	fb103StartQuiescentMode.ipDALICommunication := ipDALICommunication;
	fb103StopQuiescentMode.ipDALICommunication := ipDALICommunication;
	fb208QueryGearType.ipDALICommunication := ipDALICommunication;
	fb208QueryFeatures.ipDALICommunication := ipDALICommunication;
	fb208QuerySwitchStatus.ipDALICommunication := ipDALICommunication;
	fb208QueryDownSwitchOffThreshold.ipDALICommunication := ipDALICommunication;
	fb208QueryDownSwitchOnThreshold.ipDALICommunication := ipDALICommunication;
	fb208QueryUpSwitchOffThreshold.ipDALICommunication := ipDALICommunication;
	fb208QueryUpSwitchOnThreshold.ipDALICommunication := ipDALICommunication;
	fb208SetDownSwitchOffThreshold.ipDALICommunication := ipDALICommunication;
	fb208SetDownSwitchOnThreshold.ipDALICommunication := ipDALICommunication;
	fb208SetUpSwitchOffThreshold.ipDALICommunication := ipDALICommunication;
	fb208SetUpSwitchOnThreshold.ipDALICommunication := ipDALICommunication;
{endregion}
{region "Read"}
5:
{region "Start Qiescent Mode"}
	fb103StartQuiescentMode(bStart := TRUE,
							eAddressType := Tc3_DALI.E_DALIAddressType.Broadcast,
							eCommandPriority := Tc3_DALI.E_DALICommandPriority.Middle);
	IF (NOT fb103StartQuiescentMode.bBusy) THEN
		fb103StartQuiescentMode(bStart := FALSE);
		nStep := 10;
	END_IF
{endregion}
10:
{region "Query Gear Type"}
	fb208QueryGearType(	bStart := TRUE,
						nAddress := nAddress,
						eAddressType := Tc3_DALI.E_DALIAddressType.Short,
						eCommandPriority := Tc3_DALI.E_DALICommandPriority.Middle,
						nGearType => nGearType);
	IF (NOT fb208QueryGearType.bBusy) THEN
		fb208QueryGearType(bStart := FALSE);
		sGearType := GearType(nGearType := nGearType);
		nStep := 20;
	END_IF
{endregion}
20:
{region "Query Features"}
	fb208QueryFeatures(	bStart := TRUE,
						nAddress := nAddress,
						eAddressType := Tc3_DALI.E_DALIAddressType.Short,
						eCommandPriority := Tc3_DALI.E_DALICommandPriority.Middle);
	IF (NOT fb208QueryFeatures.bBusy) THEN
		fb208QueryFeatures(bStart := FALSE);
		bThreshold := fb208QueryFeatures.nFeatures.3;
		bAddressingPhysical := fb208QueryFeatures.nFeatures.7;
		nStep := 30;
	END_IF
{endregion}
30:
{region "Query Down Switch Off Threshold"}
	fb208QueryDownSwitchOffThreshold(	bStart := TRUE,
										nAddress := nAddress,
										eAddressType := Tc3_DALI.E_DALIAddressType.Short,
										eCommandPriority := Tc3_DALI.E_DALICommandPriority.Middle);
	IF (NOT fb208QueryDownSwitchOffThreshold.bBusy) THEN
		fb208QueryDownSwitchOffThreshold(bStart := FALSE);
		nDownSwitchOffThreshold := fb208QueryDownSwitchOffThreshold.nDownSwitchOffThreshold;
		nStep := 40;
	END_IF
{endregion}
40:
{region "Query Down Switch On Threshold"}
	fb208QueryDownSwitchOnThreshold(bStart := TRUE,
									nAddress := nAddress,
									eAddressType := Tc3_DALI.E_DALIAddressType.Short,
									eCommandPriority := Tc3_DALI.E_DALICommandPriority.Middle);
	IF (NOT fb208QueryDownSwitchOnThreshold.bBusy) THEN
		fb208QueryDownSwitchOnThreshold(bStart := FALSE);
		nDownSwitchOnThreshold := fb208QueryDownSwitchOnThreshold.nDownSwitchOnThreshold;
		nStep := 50;
	END_IF
{endregion}
50:
{region "Query Up Switch Off Threshold"}
	fb208QueryUpSwitchOffThreshold(	bStart := TRUE,
									nAddress := nAddress,
									eAddressType := Tc3_DALI.E_DALIAddressType.Short,
									eCommandPriority := Tc3_DALI.E_DALICommandPriority.Middle);
	IF (NOT fb208QueryUpSwitchOffThreshold.bBusy) THEN
		fb208QueryUpSwitchOffThreshold(bStart := FALSE);
		nUpSwitchOffThreshold := fb208QueryUpSwitchOffThreshold.nUpSwitchOffThreshold;
		nStep := 60;
	END_IF
{endregion}
60:
{region "Query Up Switch On Threshold"}
	fb208QueryUpSwitchOnThreshold(	bStart := TRUE,
									nAddress := nAddress,
									eAddressType := Tc3_DALI.E_DALIAddressType.Short,
									eCommandPriority := Tc3_DALI.E_DALICommandPriority.Middle );
	IF (NOT fb208QueryUpSwitchOnThreshold.bBusy) THEN
		fb208QueryUpSwitchOnThreshold(bStart := FALSE);
		nUpSwitchOnThreshold := fb208QueryUpSwitchOnThreshold.nUpSwitchOnThreshold;
		nStep := 70;
	END_IF
{endregion}
70:
{region "Stop Qiescent Mode"}
	fb103StopQuiescentMode(	bStart := TRUE,
							eAddressType := Tc3_DALI.E_DALIAddressType.Broadcast,
							eCommandPriority := Tc3_DALI.E_DALICommandPriority.Middle);
	IF (NOT fb103StopQuiescentMode.bBusy) THEN
		fb103StopQuiescentMode(bStart:= FALSE);
		nStep := 0;
	END_IF
{endregion}
{region "Write"}
500:
{region "Set Down Switch Off Threshold"}
	fb208SetDownSwitchOffThreshold(	bStart := TRUE,
									nAddress := nAddress,
									eAddressType := Tc3_DALI.E_DALIAddressType.Short,
									eCommandPriority := Tc3_DALI.E_DALICommandPriority.Middle,
									nDownSwitchOffThreshold := nDownSwitchOffThreshold);
	IF (NOT fb208SetDownSwitchOffThreshold.bBusy) THEN
		fb208SetDownSwitchOffThreshold(bStart := FALSE);
		nStep := 510;
	END_IF
{endregion}
510:
{region "Set Down Switch On Threshold"}
	fb208SetDownSwitchOnThreshold(	bStart := TRUE,
									nAddress := nAddress,
									eAddressType := Tc3_DALI.E_DALIAddressType.Short,
									eCommandPriority := Tc3_DALI.E_DALICommandPriority.Middle,
									nDownSwitchOnThreshold := nDownSwitchOnThreshold);
	IF (NOT fb208SetDownSwitchOnThreshold.bBusy) THEN
		fb208SetDownSwitchOnThreshold(bStart := FALSE);
		nStep := 520;
	END_IF
{endregion}
520:
{region "Set Up Switch Off Threshold"}
	fb208SetUpSwitchOffThreshold(	bStart := TRUE,
									nAddress := nAddress,
									eAddressType := Tc3_DALI.E_DALIAddressType.Short,
									eCommandPriority := Tc3_DALI.E_DALICommandPriority.Middle,
									nUpSwitchOffThreshold := nUpSwitchOffThreshold);
	IF (NOT fb208SetUpSwitchOffThreshold.bBusy) THEN
		fb208SetUpSwitchOffThreshold(bStart := FALSE);
		nStep := 530;
	END_IF
{endregion}
530:
{region "Set Up Switch On Threshold"}
	fb208SetUpSwitchOnThreshold(bStart := TRUE,
								nAddress := nAddress,
								eAddressType := Tc3_DALI.E_DALIAddressType.Short,
								eCommandPriority := Tc3_DALI.E_DALICommandPriority.Middle,
								nUpSwitchOnThreshold := nUpSwitchOnThreshold);
	IF (NOT fb208SetUpSwitchOnThreshold.bBusy) THEN
		fb208SetUpSwitchOnThreshold(bStart := FALSE);
		nStep := 0;
	END_IF
{endregion}
{endregion}
END_CASE
{endregion}

END_FUNCTION_BLOCK

// ---- POUs/DALI/PRGs/EnergyData/P_DALI_Energy_Line.TcPOU
(*
EnergyReporting reads ActiveEnergy (part 252) for all present ballasts on all (configured) DALI-lines where GVL_DALI.g_arrEnergyData[*DALI-line*,*ballast*].bHasEnergyData is TRUE.
Results are stored in GVL_DALI.g_arrEnergyData[*DALI-line*,*ballast*].fActiveEnergy. Energy Data for individual ballasts is NOT persistent.
The engergy sum per DALI-Line (Wh) and Total Energy (kWh) are persistent.

If bCheckActiveEnergy is TRUE, all present ballasts are queried for ActiveEnergy and bHasEnergyData is updated accordingly.
This will result in errors for any ballast that does not comply with part 252.
Errors will not be triggered for activations where bCheckActiveEnergy is FALSE.

After shutdown or download to PLC EnergyReporting is activated automatically internally with bCheckActiveEnergy set to TRUE

EnergyReporting is activated automatically at TOD 0:00, 6:00, 12:00, 18:00 (configurable)

NB:	The priority of commands are set to "middle" internally. Updating all lines will take a couple of minutes to finish, so be patient.
	Other critical commands on the DALI-lines take priotity.
	Add appropriate communication immediately after configuration of a new KL6821 terminal.
	That is, arrfbDALI_EnergyReporting[*DALI-Line*].ipDALICommunication := P_DALI_Background.arrfbKL6821Communication[*DALI-Line*];
*)


PROGRAM P_DALI_Energy_Line
VAR
	arrfbDALI_EnergyReporting	: ARRAY[1..SH_Light.DALI_Param.MAX_DALIV2_LINES] OF FB_DALI_EnergyReporting;
	fbDALI_EnergyDataManagement	: SH_Light.FB_DALI_EnergyDataManagement;
	nNumOfEnergyLines			: BYTE;
	bReadEnergyDataAllLines		: BOOL;
	bReportingDone				: BOOL;
	fbRTrig_ReportingDone		: R_TRIG;
	bRTrigReportingDone			: BOOL;
	
	//Task scheduling
	stLocalSystemTime 		: TIMESTRUCT;
	fbLocalSystemTime 		: FB_LocalSystemTime;
	bGetTime 				: BOOL := TRUE;
	tTimeOut 				: TIME := DEFAULT_ADS_TIMEOUT;
	bLocalSystemTimeValid	: BOOL;
	tzID       				: E_TimeZoneID := eTimeZoneID_Invalid;
	
	tdSystemTime			: TOD;
	btestTodCompare			: BOOL;
	
	
END_VAR
VAR CONSTANT
	tdMidnight						: TOD := TOD#0:0:0;
	tdMorning						: TOD := TOD#6:0:0;
	tdMidDay						: TOD := TOD#12:0:0;
	tdEvening						: TOD := TOD#18:0:0;
	tCheckDuration					: TIME:= T#5S;
	tdTestsum						: TOD := (tdMidnight + tCheckDuration);
END_VAR

VAR PERSISTENT
	arrDaliLineEnergySumWh				: ARRAY[1..SH_Light.DALI_Param.MAX_DALIV2_LINES] OF LREAL;
	fTotalEnergyWh								: LREAL;
	nMaxControlGearOperatingHours		: UINT;
END_VAR


arrfbDALI_EnergyReporting[1].ipDALICommunication := P_DALI_Background.arrfbKL6821Communication[1];
arrfbDALI_EnergyReporting[2].ipDALICommunication := P_DALI_Background.arrfbKL6821Communication[2];
arrfbDALI_EnergyReporting[3].ipDALICommunication := P_DALI_Background.arrfbKL6821Communication[3];
//arrfbDALI_EnergyReporting[4].ipDALICommunication := P_DALI_Background.arrfbKL6821Communication[4];
//arrfbDALI_EnergyReporting[5].ipDALICommunication := P_DALI_Background.arrfbKL6821Communication[5];
//arrfbDALI_EnergyReporting[6].ipDALICommunication := P_DALI_Background.arrfbKL6821Communication[6]; // for more update SH_Light.DALI_Param.MAX_DALIV2_LINES

nNumOfEnergyLines := 3;

fbLocalSystemTime(
	sNetID:= '', 
	bEnable:= bGetTime, 
	dwCycle:= 2, // cycle time (in seconds) , Synchronization  every 2 seconds.
	dwOpt:= 1, //Bit 0: If this is set, the Windows system time is additionally synchronized cyclically with the hardware clock (RTC) (corresponds to the function NT_SetTimeToRTCTime).
	tTimeout:= tTimeOut, 
	bValid=> bLocalSystemTimeValid, 
	systemTime=> stLocalSystemTime, 
	tzID=> tzID);
	
tdSystemTime := SYSTEMTIME_TO_TOD(systemTime := stLocalSystemTime);
IF	((tdSystemTime > tdMidnight AND tdSystemTime < (tdMidnight + tCheckDuration)) OR (tdSystemTime > tdMorning AND tdSystemTime < (tdMorning + tCheckDuration)) OR
	(tdSystemTime > tdMidDay AND tdSystemTime < (tdMidDay + tCheckDuration)) OR (tdSystemTime > tdEvening AND tdSystemTime < (tdEvening + tCheckDuration))) THEN
	bReadEnergyDataAllLines := TRUE;
END_IF

fbDALI_EnergyDataManagement(
	NumOfEnergyLines				:= nNumOfEnergyLines,
	bReadEnergyDataAllLines 		:= bReadEnergyDataAllLines,
	arrfbDALI_EnergyReporting		:= arrfbDALI_EnergyReporting,
	arrDaliLineEnergySum			:= arrDaliLineEnergySumWH,
	fTotalEnergyWH					:= fTotalEnergyWh,
	nMaxControlGearOperatingHours	:= nMaxControlGearOperatingHours,
	bReportingDone					=> bReportingDone
);
GVL_AHDataModbus.nTotalEnerg10kWh := TO_UINT(TRUNC(fTotalEnergyWh*EXPT(10,-4)));  //FB_DALI_EnergyDataManagement makes sure only positive values are returned. As so, conversion from REAL to UINT is appropriate
GVL_AHDataModbus.nMaxControlGearOperatingHours := nMaxControlGearOperatingHours;

END_PROGRAM

// ---- POUs/DALI/PRGs/EnergyData/P_DALI_Energy_Line_old.TcPOU
(*
EnergyReporting reads ActiveEnergy (part 252) for all present ballasts on all (configured) DALI-lines where GVL_DALI.g_arrEnergyData[*DALI-line*,*ballast*].bHasEnergyData is TRUE.
Results are stored in GVL_DALI.g_arrEnergyData[*DALI-line*,*ballast*].fActiveEnergy. Energy Data for individual ballasts is NOT persistent.
The engergy sum per DALI-Line (Wh) and Total Energy (kWh) are persistent.

If bCheckActiveEnergy is TRUE, all present ballasts are queried for ActiveEnergy and bHasEnergyData is updated accordingly.
This will result in errors for any ballast that does not comply with part 252.
Errors will not be triggered for activations where bCheckActiveEnergy is FALSE.

After shutdown or download to PLC EnergyReporting is activated automatically internally with bCheckActiveEnergy set to TRUE

EnergyReporting is activated automatically at TOD 0:00, 6:00, 12:00, 18:00 (configurable)

NB:	The priority of commands are set to "middle" internally. Updating all lines will take a couple of minutes to finish, so be patient.
	Other critical commands on the DALI-lines take priotity.
	Add appropriate communication immediately after configuration of a new KL6821 terminal.
	That is, arrfbDALI_EnergyReporting[*DALI-Line*].ipDALICommunication := P_DALI_Background.arrfbKL6821Communication[*DALI-Line*];
*)


PROGRAM P_DALI_Energy_Line_old
VAR
	arrfbDALI_EnergyReporting	: ARRAY[1..SH_Light.DALI_Param.MAX_DALIV2_LINES] OF FB_DALI_EnergyReporting_Test;
	fbDALI_EnergyDataManagement	: SH_Light.FB_DALI_EnergyDataManagement;
	nNumOfEnergyLines			: BYTE;
	bReadEnergyDataAllLines		: BOOL;
	bReportingDone				: BOOL;
	fbRTrig_ReportingDone		: R_TRIG;
	bRTrigReportingDone			: BOOL;
	
	//Task scheduling
	stLocalSystemTime 		: TIMESTRUCT;
	fbLocalSystemTime 		: FB_LocalSystemTime;
	bGetTime 				: BOOL := TRUE;
	tTimeOut 				: TIME := DEFAULT_ADS_TIMEOUT;
	bLocalSystemTimeValid	: BOOL;
	tzID       				: E_TimeZoneID := eTimeZoneID_Invalid;
	
	tdSystemTime			: TOD;
	btestTodCompare			: BOOL;
	
	
END_VAR
VAR CONSTANT
	tdMidnight						: TOD := TOD#0:0:0;
	tdMorning						: TOD := TOD#6:0:0;
	tdMidDay						: TOD := TOD#12:0:0;
	tdEvening						: TOD := TOD#18:0:0;
	tCheckDuration					: TIME:= T#5S;
	tdTestsum						: TOD := (tdMidnight + tCheckDuration);
END_VAR

VAR PERSISTENT
	arrDaliLineEnergySumWh				: ARRAY[1..SH_Light.DALI_Param.MAX_DALIV2_LINES] OF LREAL;
	nTotalEnergykWh						: UINT;
	nMaxControlGearOperatingHours		: UINT;
END_VAR


arrfbDALI_EnergyReporting[1].ipDALICommunication := P_DALI_Background.arrfbKL6821Communication[1];
arrfbDALI_EnergyReporting[2].ipDALICommunication := P_DALI_Background.arrfbKL6821Communication[2];
arrfbDALI_EnergyReporting[3].ipDALICommunication := P_DALI_Background.arrfbKL6821Communication[3];
//arrfbDALI_EnergyReporting[4].ipDALICommunication := P_DALI_Background.arrfbKL6821Communication[4];
//arrfbDALI_EnergyReporting[5].ipDALICommunication := P_DALI_Background.arrfbKL6821Communication[5];
//arrfbDALI_EnergyReporting[6].ipDALICommunication := P_DALI_Background.arrfbKL6821Communication[6]; // for more update SH_Light.DALI_Param.MAX_DALIV2_LINES

nNumOfEnergyLines := 3;

fbLocalSystemTime(
	sNetID:= '', 
	bEnable:= bGetTime, 
	dwCycle:= 2, // cycle time (in seconds) , Synchronization  every 2 seconds.
	dwOpt:= 1, //Bit 0: If this is set, the Windows system time is additionally synchronized cyclically with the hardware clock (RTC) (corresponds to the function NT_SetTimeToRTCTime).
	tTimeout:= tTimeOut, 
	bValid=> bLocalSystemTimeValid, 
	systemTime=> stLocalSystemTime, 
	tzID=> tzID);
	
tdSystemTime := SYSTEMTIME_TO_TOD(systemTime := stLocalSystemTime);
IF	((tdSystemTime > tdMidnight AND tdSystemTime < (tdMidnight + tCheckDuration)) OR (tdSystemTime > tdMorning AND tdSystemTime < (tdMorning + tCheckDuration)) OR
	(tdSystemTime > tdMidDay AND tdSystemTime < (tdMidDay + tCheckDuration)) OR (tdSystemTime > tdEvening AND tdSystemTime < (tdEvening + tCheckDuration))) THEN
	bReadEnergyDataAllLines := TRUE;
END_IF

fbDALI_EnergyDataManagement(
	NumOfEnergyLines				:= nNumOfEnergyLines,
	bReadEnergyDataAllLines 		:= bReadEnergyDataAllLines,
	arrfbDALI_EnergyReporting		:= arrfbDALI_EnergyReporting,
	arrDaliLineEnergySum			=> arrDaliLineEnergySumWH,
	nTotalEnergyKWH					=> ,
	nMaxControlGearOperatingHours	=> ,
	bDone							=> bReportingDone
);
fbRTrig_ReportingDone(CLK:=bReportingDone, Q=> bRTrigReportingDone);
IF bRTrigReportingDone THEN
	nTotalEnergykWh := fbDALI_EnergyDataManagement.nTotalEnergyKWH;
	nMaxControlGearOperatingHours:= fbDALI_EnergyDataManagement.nMaxControlGearOperatingHours;
END_IF

END_PROGRAM

// ---- POUs/EnOcean/P_EnOcean.TcPOU
PROGRAM P_EnOcean
VAR
	fbKL6581			: FB_KL6581;
	stKL6581_in  AT %I* : KL6581_INPUT;
	stKL6581_out AT %Q*	: KL6581_OUTPUT;
	stKL6581			: STR_KL6581;
	bInitCom			: BOOL := TRUE;
	
	arrEnOcean_Search	: ARRAY [1..8] OF FB_EnOcean_Search;
	nSearchIdx			: BYTE;
	bSerach				: BOOL;
	arrDevices			: ARRAY [1..8] OF INT;
	arrID				: ARRAY [1..8, 0..255] OF DWORD;
	
	
		//Trykknapper Atrium
	
	fbAtriumNiveau_Tryk_PladeB				: FB_Rec_RPS_Switch;
	fbAtriumNiveau_Tryk_Sevice				: FB_Rec_RPS_Switch;			


	//Trykknapper på gange
	fbGang_4_330_Tryk							: FB_Rec_RPS_Switch;
	
	
	//Trykknapper i rum
	fbRum_4_324_Tryk							: FB_Rec_RPS_Switch;
	fbRum_4_325_Tryk							: FB_Rec_RPS_Switch;
	fbRum_4_329_Tryk_Indgang					: FB_Rec_RPS_Switch;
	fbRum_4_329_Tryk_Ekstra						: FB_Rec_RPS_Switch;
	
    fbRum_5_339_Tryk_indgang1                   : FB_Rec_RPS_Switch;
    Rum_5_339_Tryk_Indgang2                   : FB_Rec_RPS_Switch;
    fbRum_5_341_Tryk                            : FB_Rec_RPS_Switch;
	fbRum_5_343_Tryk                            : FB_Rec_RPS_Switch;
	fbRum_5_344_Tryk                            : FB_Rec_RPS_Switch;
	fbRum_5_346_Tryk                            : FB_Rec_RPS_Switch;
	fbRum_5_345_Tryk                            : FB_Rec_RPS_Switch;
	fbRum_5_348_Tryk                            : FB_Rec_RPS_Switch;
	fbRum_5_350_Tryk                            : FB_Rec_RPS_Switch;
	fbRum_5_352_Tryk                            : FB_Rec_RPS_Switch;
	fbRum_5_353_Tryk                            : FB_Rec_RPS_Switch;
	fbRum_5_354_Tryk                            : FB_Rec_RPS_Switch;
	fbRum_5_355A_tryk_Indgang1                  : FB_Rec_RPS_Switch;
	fbRum_5_355A_Tryk_Indgang2                  : FB_Rec_RPS_Switch;
	
END_VAR

VAR CONSTANT
	byNode_1: BYTE := 1;
	byNode_2: BYTE := 2;
	byNode_3: BYTE := 3;
	byNode_4: BYTE := 4;
	byNode_5: BYTE := 5;
	byNode_6: BYTE := 6;
	byNode_7: BYTE := 7;
	byNode_8: BYTE := 8;
END_VAR


(* Kommunikation mit der KL6581. *)
(* Communication with the KL6581. *)
fbKL6581(
	bInit			:= bInitCom,
	nIdx			:= 2,
	stKL6581_in		:= stKL6581_In,
	stKL6581_out	:= stKL6581_Out,
	bReady			=> ,
	bBusy			=> ,
	bError			=> ,
	iErrorID		=> ,
	str_KL6581		=> stKL6581);
	
GVL_AHDataModbus.EnOceanError	:= TO_UINT(fbKL6581.iErrorID);

(* Warten bis der Kommunikationsbaustein initialisiert wurde.*)
(* Wait until the communication function block has been initialized. *)
IF (NOT fbKL6581.bReady) THEN
	RETURN;
END_IF

FOR nSearchIdx:= 1 TO 8 DO
	arrEnOcean_Search[nSearchIdx](
		bStart:= TRUE, 
		str_KL6581:= stKL6581 , 
		byNode:= nSearchIdx, 
		bReceive=> , 
		iDevices=>arrDevices[nSearchIdx] , 
		ar_ID=> );
		
		MEMCPY(ADR(arrID[nSearchIdx,0]), ADR(arrEnOcean_Search[nSearchIdx].ar_ID), SIZEOF(arrEnOcean_Search[nSearchIdx].ar_ID)); 
END_FOR


//A_Gang_4_330(); //Skal den fjernes, Jonas?

A_Rum_4_324();
A_Rum_4_325();
A_Rum_4_329();

A_Rum_5_339();
A_Rum_5_341();
A_Rum_5_343();
A_Rum_5_344();
A_Rum_5_345();
A_Rum_5_346();
A_Rum_5_348();
A_Rum_5_350();
A_Rum_5_352();
A_Rum_5_353();
A_Rum_5_354();
A_Rum_5_355A();
//AtriumNiveau
A_AtriumNiveau();

ACTION A_AtriumNiveau:
fbAtriumNiveau_Tryk_PladeB(
	str_KL6581:=stKL6581 , 
	byNode:=0 , 
	dw_ID:= 16#0029B92D, 
	str_EnOceanSwitch=> GVL_EnOcean.strEnOceanSwitch_AtriumNiveau_PladeB,
	by_Node=> , 
	bReceive=> );

(*fbAtriumNiveau_Tryk_Sevice(
	str_KL6581:=stKL6581 , 
	byNode:=0, 
	dw_ID:= 16#00FEE4FE87, 
	str_EnOceanSwitch=> GVL_EnOcean.strEnOceanSwitch_AtriumNiveau_Service, 
	by_Node=> , 
	bReceive=> );*)
END_ACTION

ACTION A_Gang_4_313:
fbGang_4_313_Tryk_Indgang(
	str_KL6581:=stKL6581 , 
	byNode:=byNode_2 , 
	dw_ID:= 16#0029AD03, 
	str_EnOceanSwitch=> GVL_EnOcean.strEnOceanSwitch_Gang_4_313_Indgang, 
	by_Node=> , 
	bReceive=> );
	
fbGang_4_313_Tryk_Pendler(
	str_KL6581:=stKL6581 , 
	byNode:=byNode_2 , 
	dw_ID:= 16#003C1D2B, 
	str_EnOceanSwitch=> GVL_EnOcean.strEnOceanSwitch_Gang_4_313_Pendler, 
	by_Node=> , 
	bReceive=> );
END_ACTION

ACTION A_Gang_4_330:
fbGang_4_330_Tryk(
	str_KL6581:=stKL6581 , 
	byNode:=byNode_2 , 
	dw_ID:= 16#0029B94A, 
	str_EnOceanSwitch=> GVL_EnOcean.strEnOceanSwitch_Gang_4_330, 
	by_Node=> , 
	bReceive=> );
END_ACTION

ACTION A_Rum_4_322:
fbRum_4_322_Tryk(
	str_KL6581:=stKL6581 , 
	byNode:=byNode_2 , 
	dw_ID:= 16#0029AD45, 
	str_EnOceanSwitch=> GVL_EnOcean.strEnOceanSwitch_Rum_4_322, 
	by_Node=> , 
	bReceive=> );
END_ACTION

ACTION A_Rum_4_324:
fbRum_4_324_Tryk(
	str_KL6581:=stKL6581 , 
	byNode:=byNode_2 , 
	dw_ID:= 16#00290F39, 
	str_EnOceanSwitch=> GVL_EnOcean.strEnOceanSwitch_Rum_4_324, 
	by_Node=> , 
	bReceive=> );
END_ACTION

ACTION A_Rum_4_325:
fbRum_4_325_Tryk(
	str_KL6581:=stKL6581 , 
	byNode:=byNode_2 , 
	dw_ID:= 16#00290EC6, 
	str_EnOceanSwitch=> GVL_EnOcean.strEnOceanSwitch_Rum_4_325, 
	by_Node=> , 
	bReceive=> );
END_ACTION

ACTION A_Rum_4_329:
fbRum_4_329_Tryk_Indgang(
	str_KL6581:=stKL6581 , 
	byNode:=byNode_2 , 
	dw_ID:= 16#00290EF2, 
	str_EnOceanSwitch=> GVL_EnOcean.strEnOceanSwitch_Rum_4_329_Indgang, 
	by_Node=> , 
	bReceive=> );
	
fbRum_4_329_Tryk_Ekstra(
	str_KL6581:=stKL6581 , 
	byNode:=byNode_2 , 
	dw_ID:= 16#00290ECE, 
	str_EnOceanSwitch=> GVL_EnOcean.strEnOceanSwitch_Rum_4_329_Ekstra, 
	by_Node=> , 
	bReceive=> );
END_ACTION

ACTION A_Rum_5_339:
fbRum_5_339_Tryk_Indgang1(
	str_KL6581:=stKL6581 , 
	byNode:=byNode_4 , 
	dw_ID:= 16#0029AD12, 
	str_EnOceanSwitch=> GVL_EnOcean.strEnOceanSwitch_Rum_5_339_Indgang1, 
	by_Node=> , 
	bReceive=> );

Rum_5_339_Tryk_Indgang2(
	str_KL6581:=stKL6581 , 
	byNode:=byNode_4 , 
	dw_ID:= 16#00290EDC, 
	str_EnOceanSwitch=> GVL_EnOcean.strEnOceanSwitch_Rum_5_339_Indgang2, 
	by_Node=> , 
	bReceive=> );
END_ACTION

ACTION A_Rum_5_341:
fbRum_5_341_Tryk(
	str_KL6581:=stKL6581 , 
	byNode:=byNode_2 , 
	dw_ID:= 16#00290EC5, 
	str_EnOceanSwitch=> GVL_EnOcean.strEnOceanSwitch_Rum_5_341, 
	by_Node=> , 
	bReceive=> );
END_ACTION

ACTION A_Rum_5_343:
fbRum_5_343_Tryk(
	str_KL6581:=stKL6581 , 
	byNode:=byNode_4 , 
	dw_ID:= 16#00290ECA, 
	str_EnOceanSwitch=> GVL_EnOcean.strEnOceanSwitch_Rum_5_343, 
	by_Node=> , 
	bReceive=> );
END_ACTION

ACTION A_Rum_5_344:
fbRum_5_344_Tryk(
	str_KL6581:=stKL6581 , 
	byNode:=byNode_4 , 
	dw_ID:= 16#00290EBE, 
	str_EnOceanSwitch=> GVL_EnOcean.strEnOceanSwitch_Rum_5_344, 
	by_Node=> , 
	bReceive=> );
END_ACTION

ACTION A_Rum_5_345:
fbRum_5_345_Tryk(
	str_KL6581:=stKL6581 , 
	byNode:=byNode_4 , 
	dw_ID:= 16#00290EE9, 
	str_EnOceanSwitch=> GVL_EnOcean.strEnOceanSwitch_Rum_5_345, 
	by_Node=> , 
	bReceive=> );
END_ACTION

ACTION A_Rum_5_346:
fbRum_5_346_Tryk(
	str_KL6581:=stKL6581 , 
	byNode:=byNode_4 , 
	dw_ID:= 16#00290ECD, 
	str_EnOceanSwitch=> GVL_EnOcean.strEnOceanSwitch_Rum_5_346, 
	by_Node=> , 
	bReceive=> );
END_ACTION

ACTION A_Rum_5_348:
fbRum_5_348_Tryk(
	str_KL6581:=stKL6581 , 
	byNode:=byNode_2 , 
	dw_ID:= 16#00290ED8, 
	str_EnOceanSwitch=> GVL_EnOcean.strEnOceanSwitch_Rum_5_348, 
	by_Node=> , 
	bReceive=> );
END_ACTION

ACTION A_Rum_5_350:
fbRum_5_350_Tryk(
	str_KL6581:=stKL6581 , 
	byNode:=byNode_2 , 
	dw_ID:= 16#00290F37, 
	str_EnOceanSwitch=> GVL_EnOcean.strEnOceanSwitch_Rum_5_350, 
	by_Node=> , 
	bReceive=> );
END_ACTION

ACTION A_Rum_5_352:
fbRum_5_352_Tryk(
	str_KL6581:=stKL6581 , 
	byNode:=byNode_4 , 
	dw_ID:= 16#00290EEC, 
	str_EnOceanSwitch=> GVL_EnOcean.strEnOceanSwitch_Rum_5_352, 
	by_Node=> , 
	bReceive=> );
END_ACTION

ACTION A_Rum_5_353:
fbRum_5_353_Tryk(
	str_KL6581:=stKL6581 , 
	byNode:=byNode_4 , 
	dw_ID:= 16#00290F38, 
	str_EnOceanSwitch=> GVL_EnOcean.strEnOceanSwitch_Rum_5_353, 
	by_Node=> , 
	bReceive=> );
END_ACTION

ACTION A_Rum_5_354:
fbRum_5_354_Tryk(
	str_KL6581:=stKL6581 , 
	byNode:=byNode_4 , 
	dw_ID:= 16#00290ED5, 
	str_EnOceanSwitch=> GVL_EnOcean.strEnOceanSwitch_Rum_5_354, 
	by_Node=> , 
	bReceive=> );
END_ACTION

ACTION A_Rum_5_355A:
fbRum_5_355A_Tryk_Indgang1(
	str_KL6581:=stKL6581 , 
	byNode:=byNode_4 , 
	dw_ID:= 16#003729CD, 
	str_EnOceanSwitch=> GVL_EnOcean.strEnOceanSwitch_Rum_5_355A_Indgang1, 
	by_Node=> , 
	bReceive=> );

fbRum_5_355A_Tryk_Indgang2(
	str_KL6581:=stKL6581 , 
	byNode:=byNode_4 , 
	dw_ID:= 16#0036B2B6, 
	str_EnOceanSwitch=> GVL_EnOcean.strEnOceanSwitch_Rum_5_355A_Indgang2, 
	by_Node=> , 
	bReceive=> );
END_ACTION

END_PROGRAM

// ---- POUs/MAIN.TcPOU
PROGRAM MAIN
VAR
	nAlive: INT;
	breset: BOOL;
	nDemoVariable : INT;
	nCX8200_State	AT %I*	: UINT;
END_VAR

VAR PERSISTENT
	nDemoVar_Persist: INT;
END_VAR

nAlive:= nAlive + 1;
GVL_AHDataModbus.nCX8200_State_MB := nCX8200_State;



P_SystemDK.M_nCyclic(bReset := breset );
P_DALI_DIAG();
			//P_EnOcean(); Testing fast task
DALI_Commissioning();

P_DALI_Energy_Line();

P_AHModbusComm();

//Gange
P_Gang_4_308();
P_Gang_4_330();
P_Gang_4_334A();
P_Gang_5_338();

//Rum

P_Rum_4_324();
P_Rum_4_325();
P_Rum_4_329();

P_Rum_5_339();
P_Rum_5_341();
P_Rum_5_343();
P_Rum_5_344();
P_Rum_5_345();
P_Rum_5_346();
P_Rum_5_348();
P_Rum_5_350();
P_Rum_5_350B();
P_Rum_5_352();
P_Rum_5_353();
P_Rum_5_354();

P_Rum_5_355A ();

//P_DALI_Energy_Firmware_Test();

END_PROGRAM

// ---- POUs/Tester/P_DALI2_Test.TcPOU
PROGRAM P_DALI2_Test
VAR
	fbStarCount: FB_DALI253QueryControlGearStartCounter(0);
	bStart: BOOL;
	nAddress: BYTE := 10;
	eAddressType: Tc3_DALI.E_DALIAddressType := Tc3_DALI.E_DALIAddressType.Short;
	eCommandPriority: Tc3_DALI.E_DALICommandPriority := Tc3_DALI.E_DALICommandPriority.Middle;
	nControlGearStartCounter: UDINT;
END_VAR

VAR CONSTANT
	DALI_LINE_NUM: INT := 1;
END_VAR

fbStarCount.ipDALICommunication := P_DALI_Background.arrfbKL6821Communication[DALI_LINE_NUM];


fbStarCount(
	bError=> , 
	ipResultMessage=> , 
	bStart:= bStart, 
	nAddress:= nAddress, 
	eAddressType:= eAddressType, 
	eCommandPriority:=eCommandPriority , 
	bBusy=> , 
	nControlGearStartCounter=> nControlGearStartCounter);

END_PROGRAM

// ---- GlobalTextList.TcGTLO
TEXTLIST GlobalTextList
  3955 = ' %5.2f h'
  1376 = ' %d %%'
  307 = ' %d days'
  1111 = '%2.1f  mA'
  102 = '%5.1f W'
  269 = '%5.2f h'
  621 = '%d'
  1617 = '%d %%'
  2081 = '%d days'
  3200 = '%d h'
  1372 = '%d Hz'
  2105 = '%d min'
  2025 = '%d ms'
  1540 = '%d s'
  1613 = '%d V'
  2272 = '%d weeks'
  1359 = '%d °C'
  376 = '%s'
  640 = '0'
  641 = '1'
  661 = '10'
  662 = '11'
  663 = '12'
  999 = '13'
  1000 = '14'
  1001 = '15'
  1002 = '16'
  1003 = '17'
  1004 = '18'
  1005 = '19'
  195 = '2'
  1006 = '20'
  1007 = '21'
  1008 = '22'
  1009 = '23'
  1010 = '24'
  1011 = '25'
  1012 = '26'
  1013 = '27'
  1014 = '28'
  1015 = '29'
  654 = '3'
  1016 = '30'
  1017 = '31'
  1018 = '32'
  1019 = '33'
  1020 = '34'
  1021 = '35'
  1022 = '36'
  1023 = '37'
  1024 = '38'
  1025 = '39'
  655 = '4'
  1026 = '40'
  1027 = '41'
  1028 = '42'
  1029 = '43'
  1030 = '44'
  1031 = '45'
  1032 = '46'
  1033 = '47'
  1034 = '48'
  1035 = '49'
  656 = '5'
  358 = '50'
  359 = '51'
  360 = '52'
  361 = '53'
  362 = '54'
  363 = '55'
  364 = '56'
  365 = '57'
  366 = '58'
  367 = '59'
  657 = '6'
  368 = '60'
  369 = '61'
  370 = '62'
  371 = '63'
  658 = '7'
  659 = '8'
  660 = '9'
  1089 = 'AC-supply possible'
  644 = 'Actual Level:'
  650 = 'Address Type'
  236 = 'Addressing Per Physical Selection Supported'
  1533 = 'Adjustable Emergency Level'
  1175 = 'AM Operation active:'
  1044 = 'AM operation possible'
  1045 = 'Auto Test Capability'
  1799 = 'Battery Charge'
  710 = 'Battery Duration Failure'
  3347 = 'Battery Failure'
  3316 = 'Battery Fully Charged'
  2471 = 'Bit 0'
  379 = 'Bit 1'
  2734 = 'Bit 2'
  2320 = 'Bit 3'
  929 = 'Bit 4'
  2576 = 'Bit 5'
  2065 = 'Bit 6'
  1623 = 'Bit 7'
  6 = 'Bottom Button'
  858 = 'Broadcast'
  482 = 'Button 1'
  720 = 'Button 2'
  515 = 'Button pressed'
  498 = 'Button released'
  527 = 'Button stuck / free'
  3304 = 'Cancel Hold Timer'
  2101 = 'Catch Movement'
  2319 = 'Catching:'
  897 = 'Change Addresses'
  1971 = 'Checkbox'
  372 = 'Choose group:'
  98 = 'Choose scene:'
  1571 = 'Circuit Failure'
  1173 = 'Commands'
  618 = 'Complete new installation \n(all addresses will be removed)'
  807 = 'Control'
  645 = 'Control Gear Failure:'
  445 = 'Current protection active:'
  1716 = 'Current protection device'
  668 = 'Current protection enabled:'
  5 = 'Current Protector Enabled '
  1902 = 'DALI Line:'
  1135 = 'DC-supply possible'
  560 = 'Deadtime Timer:'
  1180 = 'DI1 falling edge'
  1218 = 'DI1 rising edge'
  1726 = 'DI2 falling edge'
  1876 = 'DI2 rising edge'
  519 = 'Dim Dwn'
  63 = 'Dim Up'
  2002 = 'Dimmer Temperature'
  936 = 'Dimming Curve:'
  1317 = 'Dimming method bit 0'
  776 = 'Dimming method bit 1'
  2135 = 'Do not lock process image in case of \nDALI commands from DI1 or DI2'
  4011 = 'Double press'
  1112 = 'Double Timer Min:'
  3936 = 'Double Timer:'
  811 = 'Down'
  594 = 'Down Switch-Off Threshold'
  2357 = 'Down Switch-On Threshold'
  1482 = 'Duration Test Delay Time'
  3527 = 'Duration Test Done And Result Valid'
  3086 = 'Duration Test Failed'
  3077 = 'Duration Test Interval'
  2631 = 'Duration Test Is In Progress'
  2791 = 'Duration Test Max. Delay Exceed'
  1708 = 'Duration Test Request Pending'
  2905 = 'Duration Test Result'
  1759 = 'Emergency Lamp Failure'
  779 = 'Emergency Level'
  3733 = 'Emergency MaxLevel'
  3168 = 'Emergency Min Level'
  1204 = 'Emergency Mode'
  971 = 'Emergency Mode Active'
  1901 = 'Emergency Status'
  486 = 'Enable'
  828 = 'Enable:'
  1982 = 'EventPriority'
  32 = 'EventPriority:'
  494 = 'EventScheme'
  1113 = 'EventScheme:'
  125 = 'Extended Emergency Mode Active'
  1841 = 'Extended Fade Time only valid if Fade Time equals 0!'
  3956 = 'Extended Version'
  649 = 'Fade Running:'
  1835 = 'FadeRate'
  1844 = 'FadeTime'
  1610 = 'Failure Status'
  319 = 'Fast Fade Time:'
  2099 = 'Features'
  672 = 'Features (Read only)'
  206 = 'Features Byte 1'
  377 = 'Features Byte 2'
  2876 = 'Features Byte 3'
  3334 = 'Function Test Delay Time'
  3242 = 'Function Test Done And Result Valid'
  2712 = 'Function Test Failed'
  1801 = 'Function Test Interval'
  1945 = 'Function Test Is In Progress'
  3448 = 'Function Test Max. Delay Exceed'
  165 = 'Function Test Request Pending'
  967 = 'Gang 1.312A'
  256 = 'Gang 1.315'
  906 = 'Gang 1.316'
  207 = 'Gang 2.344'
  66 = 'Gang 2.344A'
  583 = 'Gang 2.350'
  985 = 'Gang 3.362A'
  67 = 'Gang 3.363A'
  173 = 'Gang 3.363B'
  406 = 'Gang 4.308'
  712 = 'Gang 4.310A'
  692 = 'Gang 4.313'
  459 = 'Gang 4.330'
  887 = 'Gang 4.334A'
  555 = 'Gang 4.338'
  327 = 'Gang 5.338'
  524 = 'Gang 6.310'
  316 = 'Gang 7.301'
  3204 = 'Gear Type'
  1409 = 'GearType'
  815 = 'Go to Scene'
  99 = 'Go to scene'
  852 = 'Group Address'
  2361 = 'Hardwired Inhibit Is Active'
  3553 = 'Hardwired Inhibit Supported'
  2225 = 'Hardwired Switch Is On'
  568 = 'Hold Timer:'
  199 = 'Hysteresis Min:'
  200 = 'Hysteresis:'
  790 = 'Identification Active'
  315 = 'Illuminance Level'
  37 = 'Inhibit'
  3340 = 'Inhibit Mode'
  540 = 'Input Value:'
  544 = 'Instance Error:'
  2895 = 'Instance Number:'
  3047 = 'Integral Control Gear'
  492 = 'Internal DALI power supply disabled'
  1771 = 'K-Bus Watchdog'
  3636 = 'Lamp Emergency Time'
  647 = 'Lamp Failure:'
  2812 = 'Lamp Total Operation Time'
  1521 = 'Leading Edge Mode Running'
  506 = 'LED module integrated'
  2077 = 'Linear Dimming Curve Active'
  2179 = 'Load current can be queried '
  1266 = 'Load Current Overload'
  1355 = 'Load current overload with output \nlevel reduction can be queried'
  306 = 'Load Decrease:'
  1137 = 'Load Increase:'
  2313 = 'Load over-current can be queried'
  2518 = 'Load Over-Current Shutdown'
  1226 = 'Load Rating'
  2963 = 'Load rating can be queried'
  2785 = 'Load unsuitable can be queried'
  1454 = 'Load voltage can be queried'
  516 = 'Load Voltage Out Of Limits'
  1811 = 'Lockable bytes: changeable if "Offset 2" has the Value 85 (0x55).\nFor changing use decimal value.'
  523 = 'Long press repeat'
  507 = 'Long press start'
  511 = 'Long press stop'
  43 = 'Lys Auto'
  444 = 'Lys Rum'
  489 = 'Lys Zone 1'
  2032 = 'Maintained Control Gear'
  2046 = 'Memory Bank:'
  3290 = 'Movement'
  531 = 'na'
  23 = 'Name'
  926 = 'Name of byte in memory bank'
  1038 = 'NewAddress'
  588 = 'No Movement'
  1061 = 'Non-logarithmic dimming curve can \nbe selected'
  1795 = 'Normal Mode Active'
  572 = 'Occupied'
  808 = 'Off'
  22 = 'Offset'
  1329 = 'Offset in memory bank'
  1037 = 'OldAddress'
  816 = 'On and Step Up'
  1207 = 'Open circuit detection can be queried'
  277 = 'Open Circuit:'
  1375 = 'Open Ciruit (No Load) Detect'
  619 = 'Optical feedback'
  963 = 'Output is current controlled'
  844 = 'Output regulated by current:'
  1178 = 'Parameters'
  2547 = 'Parameters Absolute Input Device'
  1580 = 'Parameters Generic Instance'
  3084 = 'Parameters LED'
  309 = 'Parameters Light Sensor'
  556 = 'Parameters Occupancy Sensor'
  465 = 'Parameters Pushbutton Sensor'
  3234 = 'Physical Selection Supported'
  1847 = 'Physical selection supported'
  708 = 'PIR'
  457 = 'PIR status'
  1071 = 'Please check if Current Protector is present \nby reading parameters first.'
  308 = 'Please select the desired Short Address in the table above.'
  1458 = 'Please select the function you need from dropdown above'
  751 = 'Position Event'
  245 = 'Possible Operating Modes'
  719 = 'Power pulse operation'
  1744 = 'Power supply integrated'
  1561 = 'PP Operation active:'
  2321 = 'Prolong Time (30sec / Step)'
  970 = 'PWM Operation active:'
  1882 = 'PWM operation possible'
  1487 = 'Query idle time detection \nenabled'
  701 = 'Query load decrease enabled'
  1351 = 'Query load increase enabled'
  837 = 'Query reduction luminous flux \nregarding thermal overload'
  463 = 'Query short circuit enabled'
  1293 = 'Query thermal switch enabled'
  617 = 'Random Addressing'
  2174 = 'Rated Duration'
  881 = 'Re-Light / Reset Inhibit'
  373 = 'Read'
  1611 = 'Read Only'
  1531 = 'Reads all Fading Parameters'
  768 = 'Real Load Power'
  854 = 'Real load power can be queried'
  810 = 'Recall Max Level'
  809 = 'Recall Min Level'
  186 = 'Ref. Measurement failed:'
  439 = 'Reference System Power'
  2713 = 'Relight Rest Mode Supported'
  580 = 'Repeat'
  470 = 'Repeat Timer:'
  1913 = 'Report Timer:'
  716 = 'Reset Duration Test Done Flag'
  592 = 'Reset Function Test Done Flag'
  2418 = 'Reset inactive process image'
  3150 = 'Reset Lamp Time'
  648 = 'Reset State:'
  2888 = 'Resolution:'
  299 = 'Rest'
  591 = 'Rest Mode Active'
  2001 = 'RMS Load Current'
  784 = 'RMS Load Voltage'
  586 = 'RMS Supply Voltage'
  874 = 'Rum 1.106'
  65 = 'Rum 1.108'
  175 = 'Rum 1.111A'
  924 = 'Rum 1.111C'
  219 = 'Rum 1.111D'
  690 = 'Rum 1.111E'
  912 = 'Rum 1.115'
  126 = 'Rum 1.118'
  215 = 'Rum 1.312A'
  725 = 'Rum 1.318'
  839 = 'Rum 1.319'
  456 = 'Rum 1.320'
  800 = 'Rum 1.321'
  622 = 'Rum 1.322'
  646 = 'Rum 1.323'
  966 = 'Rum 1.324'
  95 = 'Rum 1.325'
  335 = 'Rum 1.326'
  150 = 'Rum 1.327'
  651 = 'Rum 1.328'
  980 = 'Rum 1.330'
  262 = 'Rum 1115'
  642 = 'Rum 2.341'
  978 = 'Rum 2.345'
  736 = 'Rum 2.349'
  593 = 'Rum 2.351'
  122 = 'Rum 2.352'
  27 = 'Rum 2.353'
  41 = 'Rum 2.354'
  697 = 'Rum 2.355'
  826 = 'Rum 2.356'
  561 = 'Rum 2.357'
  952 = 'Rum 3.329'
  623 = 'Rum 3_329'
  174 = 'Rum 4.307'
  166 = 'Rum 4.311'
  870 = 'Rum 4.313'
  584 = 'Rum 4.316'
  812 = 'Rum 4.317'
  458 = 'Rum 4.321'
  565 = 'Rum 4.322'
  803 = 'Rum 4.324'
  201 = 'Rum 4.325'
  251 = 'Rum 4.329'
  795 = 'Rum 5.354'
  19 = 'Rum 5_345'
  15 = 'Rum 5_352'
  693 = 'Rum 5_354'
  1093 = 'Rum 5_355A'
  430 = 'Rum 6.310 Sofagruppe'
  348 = 'Rum 6.327'
  891 = 'Rum 6.328'
  11 = 'Rum 6.329'
  72 = 'Rum 6.330B'
  197 = 'Rum 6.331'
  564 = 'Rum 6.333'
  997 = 'Rum 6.337'
  31 = 'Rum 6_330A'
  616 = 'Scan devices by address'
  1036 = 'Scene Level'
  814 = 'Scene:'
  1366 = 'Set Extended Fade Time'
  252 = 'Set Fade Rate'
  1875 = 'Set Fade Time'
  846 = 'Short Address'
  1861 = 'Short Address Range'
  1041 = 'Short Address:'
  34 = 'Short Circuit:'
  503 = 'Short press'
  1516 = 'Short Timer Min:'
  478 = 'Short Timer:'
  2548 = 'Shutdown Invalid Dimming Method'
  1852 = 'Single Short Address'
  395 = 'SP_Lux: %.0f'
  525 = 'SP_Lux: %f'
  615 = 'Start'
  582 = 'Start Duration Test'
  2374 = 'Start Function Test'
  155 = 'Start Identification'
  620 = 'Start with address:'
  2346 = 'State Incandescent Lamp'
  643 = 'Status'
  958 = 'Status Absolute Input Device'
  2506 = 'Status Generic Instance'
  3076 = 'Status LED'
  317 = 'Status Light Sensor'
  597 = 'Status Occupancy Sensor'
  536 = 'Status Pushbutton Sensor'
  558 = 'Step Down'
  813 = 'Step Down and Off'
  818 = 'Step Up'
  1193 = 'Stop Test'
  164 = 'Stuck Timer:'
  1256 = 'Supply Frequency'
  2271 = 'Supply frequency can be queried'
  1975 = 'Supply Frequency Out of Limits'
  2505 = 'Supply voltage can be queried'
  2707 = 'Supply Voltage Out Of Limits'
  1042 = 'Switch Off'
  375 = 'Switch On'
  3781 = 'Switched Maintained Control Gear'
  2168 = 'Temperature can be queried'
  2458 = 'Terminal Event'
  1848 = 'Test Execution Timeout'
  849 = 'Test Type A'
  2013 = 'Thermal Overload'
  2042 = 'Thermal Overload with output\nlevel reduction can be queried'
  1108 = 'Thermal Overload:'
  355 = 'Thermal Shut Down:'
  2507 = 'Thermal Shutdown'
  2226 = 'Thermal Shutdown can be queried'
  2733 = 'Threshold Editable'
  305 = 'To'
  973 = 'Top Button'
  136 = 'Trailing Edge ModeRunning'
  864 = 'Unaddressed'
  817 = 'Up'
  3123 = 'Up Switch-Off Threshold'
  1449 = 'Up Switch-On Threshold'
  2521 = 'V%s'
  576 = 'Vacant'
  1205 = 'Value'
  24 = 'Value Dec'
  1435 = 'Value decimal'
  25 = 'Value Hex'
  2231 = 'Value hexadecimal,\nto change use\nvalue decimal'
  374 = 'Write'
  2104 = 'Write\nDimming Curve'
  1047 = 'Write default values'
  490 = 'Write parameters'
END_TEXTLIST

// ---- POUs/Alle_Rum/Gange/Gang_4_334A/Visualization_4_334A.TcVIS
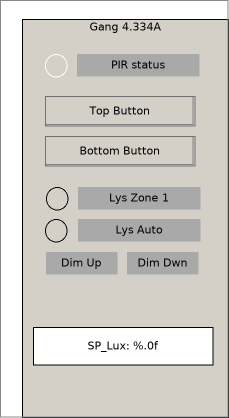
VISUALIZATION Visualization_4_334A  // 229x418
    RoundedRectangle (22,19 207x399), "Gang 4.334A"
    Rectangle (33,327 180x38), "SP_Lux: %.0f", text variable: P_Gang_4_334A.fbLys.fbLightCtrl.fLuxZone1
    Button (45,96 150x30), "Top Button"
        tap P_Gang_4_334A.bTopButtonZone1_Visu
    Button (45,136 150x30), "Bottom Button"
        tap P_Gang_4_334A.bBottomButtonZone1_Visu
    Ellipse (46,187 22x23), colour toggle: P_Gang_4_334A.fbLys.fbLightCtrl.bOnZone1
    Rectangle (78,187 122x22), "Lys Zone 1"
    Rectangle (46,252 71x22), "Dim Up", colour toggle: P_Gang_4_334A.fbLys.fbLightCtrl.bDimUp
    Rectangle (127,252 71x22), "Dim Dwn", colour toggle: P_Gang_4_334A.fbLys.fbLightCtrl.bDimDwn
    Ellipse (45,219 22x23), colour toggle: P_Gang_4_334A.fbLys.fbLightCtrl.bAutoZone1
    Rectangle (78,219 122x22), "Lys Auto"
    Ellipse (45,54 22x23), colour toggle: P_Gang_4_334A.fbLys.fbLightCtrl.bPIR
    Rectangle (77,54 122x22), "PIR status"
END_VISUALIZATION

// ---- POUs/Alle_Rum/Gange/Gang_4_330/Visualization_4_330.TcVIS
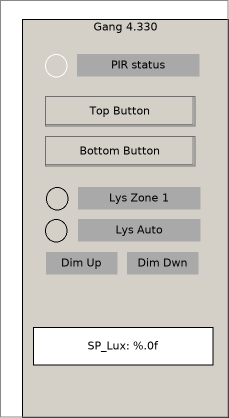
VISUALIZATION Visualization_4_330  // 229x418
    RoundedRectangle (22,19 207x399), "Gang 4.330"
    Rectangle (33,327 180x38), "SP_Lux: %.0f", text variable: P_Gang_4_330.arrfbLysGruppe[1].fbLightCtrl.fLuxZone1
    Button (45,96 150x30), "Top Button"
        tap P_Gang_4_330.bTopButtonZone1_Visu
    Button (45,136 150x30), "Bottom Button"
        tap P_Gang_4_330.bBottomButtonZone1_Visu
    Ellipse (46,187 22x23), colour toggle: P_Gang_4_330.fbLys.fbLightCtrl.bOnZone1
    Rectangle (78,187 122x22), "Lys Zone 1"
    Rectangle (46,252 71x22), "Dim Up", colour toggle: P_Gang_4_330.arrfbLysGruppe[1].fbLightCtrl.bDimUp
    Rectangle (127,252 71x22), "Dim Dwn", colour toggle: P_Gang_4_330.arrfbLysGruppe[1].fbLightCtrl.bDimDwn
    Ellipse (45,219 22x23), colour toggle: P_Gang_4_330.arrfbLysGruppe[1].fbLightCtrl.bAutoZone1
    Rectangle (78,219 122x22), "Lys Auto"
    Ellipse (45,54 22x23), colour toggle: P_Gang_4_330.arrfbLysGruppe[1].fbLightCtrl.bPIR
    Rectangle (77,54 122x22), "PIR status"
END_VISUALIZATION

// ---- POUs/Alle_Rum/Gange/1Gang_4_310A/Visualization_4_310A.TcVIS
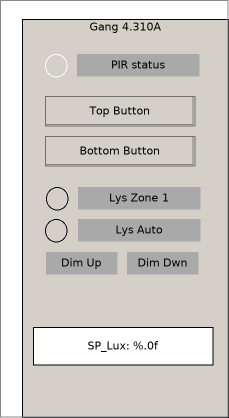
VISUALIZATION Visualization_4_310A  // 229x418
    RoundedRectangle (22,19 207x399), "Gang 4.310A"
    Rectangle (33,327 180x38), "SP_Lux: %.0f", text variable: P_Gang_4_310A.fbLys.fbLightCtrl.fLuxZone1
    Button (45,96 150x30), "Top Button"
        tap P_Gang_4_310A.bTopButtonZone1_Visu
    Button (45,136 150x30), "Bottom Button"
        tap P_Gang_4_310A.bBottomButtonZone1_Visu
    Ellipse (46,187 22x23), colour toggle: P_Gang_4_310A.fbLys.fbLightCtrl.bOnZone1
    Rectangle (78,187 122x22), "Lys Zone 1"
    Rectangle (46,252 71x22), "Dim Up", colour toggle: P_Gang_4_310A.fbLys.fbLightCtrl.bDimUp
    Rectangle (127,252 71x22), "Dim Dwn", colour toggle: P_Gang_4_310A.fbLys.fbLightCtrl.bDimDwn
    Ellipse (45,219 22x23), colour toggle: P_Gang_4_310A.fbLys.fbLightCtrl.bAutoZone1
    Rectangle (78,219 122x22), "Lys Auto"
    Ellipse (45,54 22x23), colour toggle: P_Gang_4_310A.fbLys.fbLightCtrl.bPIR
    Rectangle (77,54 122x22), "PIR status"
END_VISUALIZATION

// ---- POUs/Alle_Rum/Gange/Gang_4_308/Visualization_4_308.TcVIS
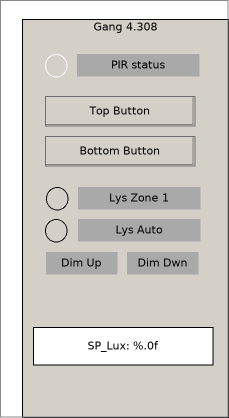
VISUALIZATION Visualization_4_308  // 229x418
    RoundedRectangle (22,19 207x399), "Gang 4.308"
    Rectangle (33,327 180x38), "SP_Lux: %.0f", text variable: P_Gang_4_308.arrfbLysGruppe[1].fbLightCtrl.fLuxZone1
    Button (45,96 150x30), "Top Button"
        tap P_Gang_4_308.bTopButtonZone1_Visu
    Button (45,136 150x30), "Bottom Button"
        tap P_Gang_4_308.bBottomButtonZone1_Visu
    Ellipse (46,187 22x23), colour toggle: P_Gang_4_308.arrfbLysGruppe[1].fbLightCtrl.bOnZone1
    Rectangle (78,187 122x22), "Lys Zone 1"
    Rectangle (46,252 71x22), "Dim Up", colour toggle: P_Gang_4_308.arrfbLysGruppe[1].fbLightCtrl.bDimUp
    Rectangle (127,252 71x22), "Dim Dwn", colour toggle: P_Gang_4_308.arrfbLysGruppe[1].fbLightCtrl.bDimDwn
    Ellipse (45,219 22x23), colour toggle: P_Gang_4_308.arrfbLysGruppe[1].fbLightCtrl.bAutoZone1
    Rectangle (78,219 122x22), "Lys Auto"
    Ellipse (45,54 22x23), colour toggle: P_Gang_4_308.arrfbLysGruppe[1].fbLightCtrl.bPIR
    Rectangle (77,54 122x22), "PIR status"
END_VISUALIZATION

// ---- POUs/Alle_Rum/Rum_Med_DALI_Pir/Rum_4_325/Visualization_4_324_1.TcVIS
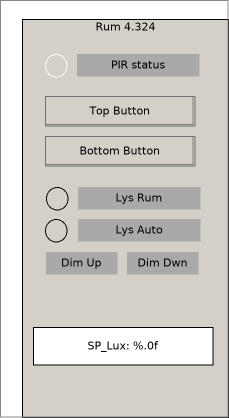
VISUALIZATION Visualization_4_324_1  // 229x418
    RoundedRectangle (22,19 207x399), "Rum 4.324"
    Rectangle (33,327 180x38), "SP_Lux: %.0f", text variable: P_Rum_4_324.fbLys.fbLightCtrl.fLuxZone1
    Button (45,96 150x30), "Top Button"
        tap P_Rum_4_324.bTopButtonZone1_Visu
    Button (45,136 150x30), "Bottom Button"
        tap P_Rum_4_324.bBottomButtonZone1_Visu
    Ellipse (46,187 22x23), colour toggle: P_Rum_4_324.fbLys.fbLightCtrl.bOnZone1
    Rectangle (78,187 122x22), "Lys Rum"
    Rectangle (46,252 71x22), "Dim Up", colour toggle: P_Rum_4_324.fbLys.fbLightCtrl.bDimUp
    Rectangle (127,252 71x22), "Dim Dwn", colour toggle: P_Rum_4_324.fbLys.fbLightCtrl.bDimDwn
    Ellipse (45,219 22x23), colour toggle: P_Rum_4_324.fbLys.fbLightCtrl.bAutoZone1
    Rectangle (78,219 122x22), "Lys Auto"
    Ellipse (45,54 22x23), colour toggle: P_Rum_4_324.fbLys.fbLightCtrl.bPIR
    Rectangle (77,54 122x22), "PIR status"
END_VISUALIZATION

// ---- POUs/Alle_Rum/Rum_Med_DALI_Pir/Rum_5_339/Visualization_5_352_1_1_1_2_2.TcVIS
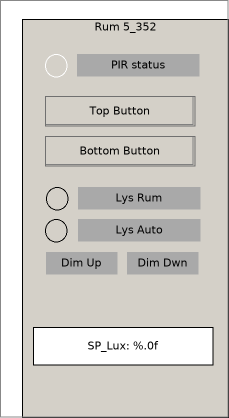
VISUALIZATION Visualization_5_352_1_1_1_2_2  // 229x418
    RoundedRectangle (22,19 207x399), "Rum 5_352"
    Rectangle (33,327 180x38), "SP_Lux: %.0f", text variable: P_Rum_4_324.fbLys.fbLightCtrl.fLuxZone1
    Button (45,96 150x30), "Top Button"
        tap P_Rum_5_352.bTopButtonZone1_Visu
    Button (45,136 150x30), "Bottom Button"
        tap P_Rum_5_352.bBottomButtonZone1_Visu
    Ellipse (46,187 22x23), colour toggle: P_Rum_5_352.fbLys.fbLightCtrl.bOnZone1
    Rectangle (78,187 122x22), "Lys Rum"
    Rectangle (46,252 71x22), "Dim Up", colour toggle: P_Rum_5_352.fbLys.fbLightCtrl.bDimUp
    Rectangle (127,252 71x22), "Dim Dwn", colour toggle: P_Rum_5_352.fbLys.fbLightCtrl.bDimDwn
    Ellipse (45,219 22x23), colour toggle: P_Rum_5_352.fbLys.fbLightCtrl.bAutoZone1
    Rectangle (78,219 122x22), "Lys Auto"
    Ellipse (45,54 22x23), colour toggle: P_Rum_5_352.fbLys.fbLightCtrl.bPIR
    Rectangle (77,54 122x22), "PIR status"
END_VISUALIZATION

// ---- POUs/Alle_Rum/Rum_Med_DALI_Pir/Rum_5_343/Visualization_5_352_1_1_1_2_1.TcVIS
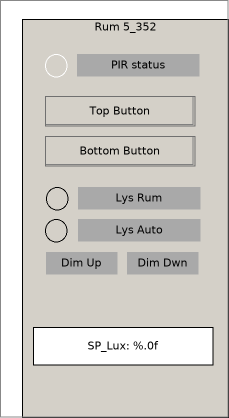
VISUALIZATION Visualization_5_352_1_1_1_2_1  // 229x418
    RoundedRectangle (22,19 207x399), "Rum 5_352"
    Rectangle (33,327 180x38), "SP_Lux: %.0f", text variable: P_Rum_4_324.fbLys.fbLightCtrl.fLuxZone1
    Button (45,96 150x30), "Top Button"
        tap P_Rum_5_352.bTopButtonZone1_Visu
    Button (45,136 150x30), "Bottom Button"
        tap P_Rum_5_352.bBottomButtonZone1_Visu
    Ellipse (46,187 22x23), colour toggle: P_Rum_5_352.fbLys.fbLightCtrl.bOnZone1
    Rectangle (78,187 122x22), "Lys Rum"
    Rectangle (46,252 71x22), "Dim Up", colour toggle: P_Rum_5_352.fbLys.fbLightCtrl.bDimUp
    Rectangle (127,252 71x22), "Dim Dwn", colour toggle: P_Rum_5_352.fbLys.fbLightCtrl.bDimDwn
    Ellipse (45,219 22x23), colour toggle: P_Rum_5_352.fbLys.fbLightCtrl.bAutoZone1
    Rectangle (78,219 122x22), "Lys Auto"
    Ellipse (45,54 22x23), colour toggle: P_Rum_5_352.fbLys.fbLightCtrl.bPIR
    Rectangle (77,54 122x22), "PIR status"
END_VISUALIZATION

// ---- POUs/Alle_Rum/Rum_Med_DALI_Pir/Rum_5_346/Visualization_5_352_1_1_1_1.TcVIS
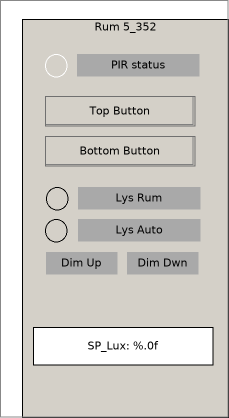
VISUALIZATION Visualization_5_352_1_1_1_1  // 229x418
    RoundedRectangle (22,19 207x399), "Rum 5_352"
    Rectangle (33,327 180x38), "SP_Lux: %.0f", text variable: P_Rum_4_324.fbLys.fbLightCtrl.fLuxZone1
    Button (45,96 150x30), "Top Button"
        tap P_Rum_5_352.bTopButtonZone1_Visu
    Button (45,136 150x30), "Bottom Button"
        tap P_Rum_5_352.bBottomButtonZone1_Visu
    Ellipse (46,187 22x23), colour toggle: P_Rum_5_352.fbLys.fbLightCtrl.bOnZone1
    Rectangle (78,187 122x22), "Lys Rum"
    Rectangle (46,252 71x22), "Dim Up", colour toggle: P_Rum_5_352.fbLys.fbLightCtrl.bDimUp
    Rectangle (127,252 71x22), "Dim Dwn", colour toggle: P_Rum_5_352.fbLys.fbLightCtrl.bDimDwn
    Ellipse (45,219 22x23), colour toggle: P_Rum_5_352.fbLys.fbLightCtrl.bAutoZone1
    Rectangle (78,219 122x22), "Lys Auto"
    Ellipse (45,54 22x23), colour toggle: P_Rum_5_352.fbLys.fbLightCtrl.bPIR
    Rectangle (77,54 122x22), "PIR status"
END_VISUALIZATION

// ---- POUs/Alle_Rum/Rum_Med_DALI_Pir/Rum_5_348/Visualization_5_352_1_1.TcVIS
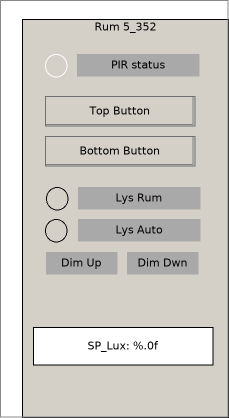
VISUALIZATION Visualization_5_352_1_1  // 229x418
    RoundedRectangle (22,19 207x399), "Rum 5_352"
    Rectangle (33,327 180x38), "SP_Lux: %.0f", text variable: P_Rum_4_324.fbLys.fbLightCtrl.fLuxZone1
    Button (45,96 150x30), "Top Button"
        tap P_Rum_5_352.bTopButtonZone1_Visu
    Button (45,136 150x30), "Bottom Button"
        tap P_Rum_5_352.bBottomButtonZone1_Visu
    Ellipse (46,187 22x23), colour toggle: P_Rum_5_352.fbLys.fbLightCtrl.bOnZone1
    Rectangle (78,187 122x22), "Lys Rum"
    Rectangle (46,252 71x22), "Dim Up", colour toggle: P_Rum_5_352.fbLys.fbLightCtrl.bDimUp
    Rectangle (127,252 71x22), "Dim Dwn", colour toggle: P_Rum_5_352.fbLys.fbLightCtrl.bDimDwn
    Ellipse (45,219 22x23), colour toggle: P_Rum_5_352.fbLys.fbLightCtrl.bAutoZone1
    Rectangle (78,219 122x22), "Lys Auto"
    Ellipse (45,54 22x23), colour toggle: P_Rum_5_352.fbLys.fbLightCtrl.bPIR
    Rectangle (77,54 122x22), "PIR status"
END_VISUALIZATION

// ---- POUs/Alle_Rum/Rum_Med_DALI_Pir/Rum_5_344/Visualization_5_352_1_1_1.TcVIS
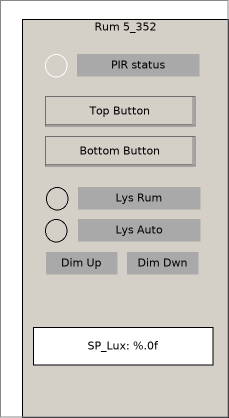
VISUALIZATION Visualization_5_352_1_1_1  // 229x418
    RoundedRectangle (22,19 207x399), "Rum 5_352"
    Rectangle (33,327 180x38), "SP_Lux: %.0f", text variable: P_Rum_4_324.fbLys.fbLightCtrl.fLuxZone1
    Button (45,96 150x30), "Top Button"
        tap P_Rum_5_352.bTopButtonZone1_Visu
    Button (45,136 150x30), "Bottom Button"
        tap P_Rum_5_352.bBottomButtonZone1_Visu
    Ellipse (46,187 22x23), colour toggle: P_Rum_5_352.fbLys.fbLightCtrl.bOnZone1
    Rectangle (78,187 122x22), "Lys Rum"
    Rectangle (46,252 71x22), "Dim Up", colour toggle: P_Rum_5_352.fbLys.fbLightCtrl.bDimUp
    Rectangle (127,252 71x22), "Dim Dwn", colour toggle: P_Rum_5_352.fbLys.fbLightCtrl.bDimDwn
    Ellipse (45,219 22x23), colour toggle: P_Rum_5_352.fbLys.fbLightCtrl.bAutoZone1
    Rectangle (78,219 122x22), "Lys Auto"
    Ellipse (45,54 22x23), colour toggle: P_Rum_5_352.fbLys.fbLightCtrl.bPIR
    Rectangle (77,54 122x22), "PIR status"
END_VISUALIZATION

// ---- POUs/Alle_Rum/Rum_Med_DALI_Pir/Rum_5_352/Visualization_5_352.TcVIS
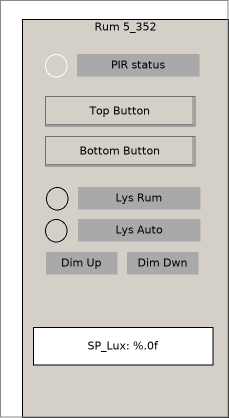
VISUALIZATION Visualization_5_352  // 229x418
    RoundedRectangle (22,19 207x399), "Rum 5_352"
    Rectangle (33,327 180x38), "SP_Lux: %.0f", text variable: P_Rum_4_324.fbLys.fbLightCtrl.fLuxZone1
    Button (45,96 150x30), "Top Button"
        tap P_Rum_5_352.bTopButtonZone1_Visu
    Button (45,136 150x30), "Bottom Button"
        tap P_Rum_5_352.bBottomButtonZone1_Visu
    Ellipse (46,187 22x23), colour toggle: P_Rum_5_352.fbLys.fbLightCtrl.bOnZone1
    Rectangle (78,187 122x22), "Lys Rum"
    Rectangle (46,252 71x22), "Dim Up", colour toggle: P_Rum_5_352.fbLys.fbLightCtrl.bDimUp
    Rectangle (127,252 71x22), "Dim Dwn", colour toggle: P_Rum_5_352.fbLys.fbLightCtrl.bDimDwn
    Ellipse (45,219 22x23), colour toggle: P_Rum_5_352.fbLys.fbLightCtrl.bAutoZone1
    Rectangle (78,219 122x22), "Lys Auto"
    Ellipse (45,54 22x23), colour toggle: P_Rum_5_352.fbLys.fbLightCtrl.bPIR
    Rectangle (77,54 122x22), "PIR status"
END_VISUALIZATION

// ---- POUs/Alle_Rum/Rum_Med_DALI_Pir/Rum_4_329/Visualization_4_329.TcVIS
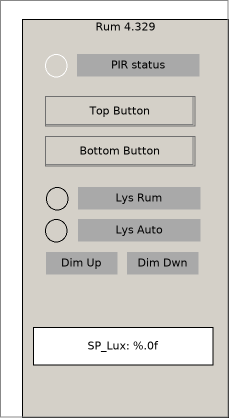
VISUALIZATION Visualization_4_329  // 229x418
    RoundedRectangle (22,19 207x399), "Rum 4.329"
    Rectangle (33,327 180x38), "SP_Lux: %.0f", text variable: P_Rum_4_329.fbLys.fbLightCtrl.fLuxZone1
    Button (45,96 150x30), "Top Button"
        tap P_Rum_4_329.bTopButtonZone1_Visu
    Button (45,136 150x30), "Bottom Button"
        tap P_Rum_4_329.bBottomButtonZone1_Visu
    Ellipse (46,187 22x23), colour toggle: P_Rum_4_329.fbLys.fbLightCtrl.bOnZone1
    Rectangle (78,187 122x22), "Lys Rum"
    Rectangle (46,252 71x22), "Dim Up", colour toggle: P_Rum_4_329.fbLys.fbLightCtrl.bDimUp
    Rectangle (127,252 71x22), "Dim Dwn", colour toggle: P_Rum_4_329.fbLys.fbLightCtrl.bDimDwn
    Ellipse (45,219 22x23), colour toggle: P_Rum_4_329.fbLys.fbLightCtrl.bAutoZone1
    Rectangle (78,219 122x22), "Lys Auto"
    Ellipse (45,54 22x23), colour toggle: P_Rum_4_329.fbLys.fbLightCtrl.bPIR
    Rectangle (77,54 122x22), "PIR status"
END_VISUALIZATION

// ---- POUs/Alle_Rum/Rum_Med_DALI_Pir/1Rum_4_307/Visualization_4_307.TcVIS
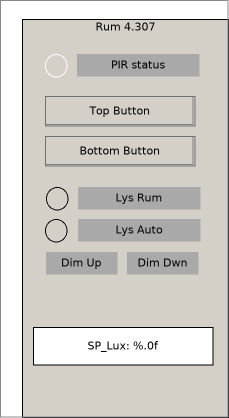
VISUALIZATION Visualization_4_307  // 229x418
    RoundedRectangle (22,19 207x399), "Rum 4.307"
    Rectangle (33,327 180x38), "SP_Lux: %.0f", text variable: P_Rum_4_307.fbLys.fbLightCtrl.fLuxZone1
    Button (45,96 150x30), "Top Button"
        tap P_Rum_4_307.bTopButtonZone1_Visu
    Button (45,136 150x30), "Bottom Button"
        tap P_Rum_4_307.bBottomButtonZone1_Visu
    Ellipse (46,187 22x23), colour toggle: P_Rum_4_307.fbLys.fbLightCtrl.bOnZone1
    Rectangle (78,187 122x22), "Lys Rum"
    Rectangle (46,252 71x22), "Dim Up", colour toggle: P_Rum_4_307.fbLys.fbLightCtrl.bDimUp
    Rectangle (127,252 71x22), "Dim Dwn", colour toggle: P_Rum_4_307.fbLys.fbLightCtrl.bDimDwn
    Ellipse (45,219 22x23), colour toggle: P_Rum_4_307.fbLys.fbLightCtrl.bAutoZone1
    Rectangle (78,219 122x22), "Lys Auto"
    Ellipse (45,54 22x23), colour toggle: P_Rum_4_307.fbLys.fbLightCtrl.bPIR
    Rectangle (77,54 122x22), "PIR status"
END_VISUALIZATION

// ---- POUs/Alle_Rum/Rum_Med_DALI_Pir/1Rum_4_313/Visualization_4_313.TcVIS
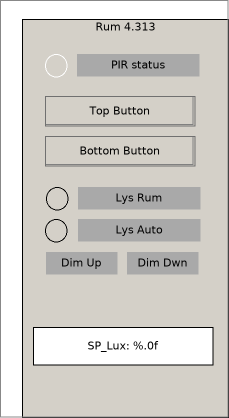
VISUALIZATION Visualization_4_313  // 229x418
    RoundedRectangle (22,19 207x399), "Rum 4.313"
    Rectangle (33,327 180x38), "SP_Lux: %.0f", text variable: P_Rum_4_313.fbLys.fbLightCtrl.fLuxZone1
    Button (45,96 150x30), "Top Button"
        tap P_Rum_4_313.bTopButtonZone1_Visu
    Button (45,136 150x30), "Bottom Button"
        tap P_Rum_4_313.bBottomButtonZone1_Visu
    Ellipse (46,187 22x23), colour toggle: P_Rum_4_313.fbLys.fbLightCtrl.bOnZone1
    Rectangle (78,187 122x22), "Lys Rum"
    Rectangle (46,252 71x22), "Dim Up", colour toggle: P_Rum_4_313.fbLys.fbLightCtrl.bDimUp
    Rectangle (127,252 71x22), "Dim Dwn", colour toggle: P_Rum_4_313.fbLys.fbLightCtrl.bDimDwn
    Ellipse (45,219 22x23), colour toggle: P_Rum_4_313.fbLys.fbLightCtrl.bAutoZone1
    Rectangle (78,219 122x22), "Lys Auto"
    Ellipse (45,54 22x23), colour toggle: P_Rum_4_313.fbLys.fbLightCtrl.bPIR
    Rectangle (77,54 122x22), "PIR status"
END_VISUALIZATION

// ---- POUs/Alle_Rum/Rum_Med_DALI_Pir/1Rum_4_316/Visualization_4_316.TcVIS
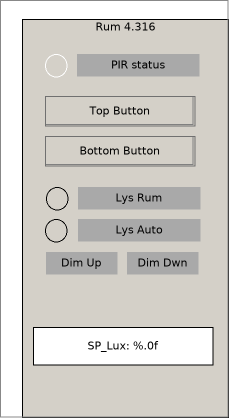
VISUALIZATION Visualization_4_316  // 229x418
    RoundedRectangle (22,19 207x399), "Rum 4.316"
    Rectangle (33,327 180x38), "SP_Lux: %.0f", text variable: P_Rum_4_316.fbLys.fbLightCtrl.fLuxZone1
    Button (45,96 150x30), "Top Button"
        tap P_Rum_4_316.bTopButtonZone1_Visu
    Button (45,136 150x30), "Bottom Button"
        tap P_Rum_4_316.bBottomButtonZone1_Visu
    Ellipse (46,187 22x23), colour toggle: P_Rum_4_316.fbLys.fbLightCtrl.bOnZone1
    Rectangle (78,187 122x22), "Lys Rum"
    Rectangle (46,252 71x22), "Dim Up", colour toggle: P_Rum_4_316.fbLys.fbLightCtrl.bDimUp
    Rectangle (127,252 71x22), "Dim Dwn", colour toggle: P_Rum_4_316.fbLys.fbLightCtrl.bDimDwn
    Ellipse (45,219 22x23), colour toggle: P_Rum_4_316.fbLys.fbLightCtrl.bAutoZone1
    Rectangle (78,219 122x22), "Lys Auto"
    Ellipse (45,54 22x23), colour toggle: P_Rum_4_316.fbLys.fbLightCtrl.bPIR
    Rectangle (77,54 122x22), "PIR status"
END_VISUALIZATION

// ---- POUs/Alle_Rum/Rum_Med_DALI_Pir/1Rum_4_321/Visualization_4_321.TcVIS
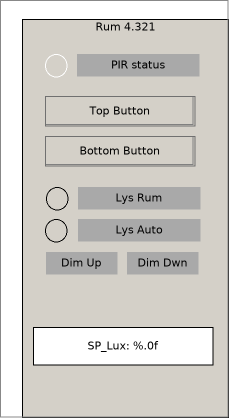
VISUALIZATION Visualization_4_321  // 229x418
    RoundedRectangle (22,19 207x399), "Rum 4.321"
    Rectangle (33,327 180x38), "SP_Lux: %.0f", text variable: P_Rum_4_321.fbLys.fbLightCtrl.fLuxZone1
    Button (45,96 150x30), "Top Button"
        tap P_Rum_4_321.bTopButtonZone1_Visu
    Button (45,136 150x30), "Bottom Button"
        tap P_Rum_4_321.bBottomButtonZone1_Visu
    Ellipse (46,187 22x23), colour toggle: P_Rum_4_321.fbLys.fbLightCtrl.bOnZone1
    Rectangle (78,187 122x22), "Lys Rum"
    Rectangle (46,252 71x22), "Dim Up", colour toggle: P_Rum_4_321.fbLys.fbLightCtrl.bDimUp
    Rectangle (127,252 71x22), "Dim Dwn", colour toggle: P_Rum_4_321.fbLys.fbLightCtrl.bDimDwn
    Ellipse (45,219 22x23), colour toggle: P_Rum_4_321.fbLys.fbLightCtrl.bAutoZone1
    Rectangle (78,219 122x22), "Lys Auto"
    Ellipse (45,54 22x23), colour toggle: P_Rum_4_321.fbLys.fbLightCtrl.bPIR
    Rectangle (77,54 122x22), "PIR status"
END_VISUALIZATION

// ---- POUs/Alle_Rum/Rum_Med_DALI_Pir/1Rum_4_322/Visualization_4_322.TcVIS
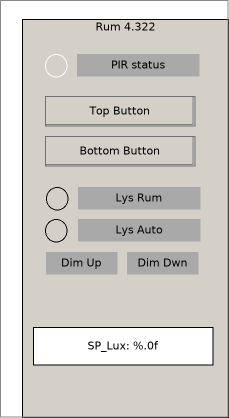
VISUALIZATION Visualization_4_322  // 229x418
    RoundedRectangle (22,19 207x399), "Rum 4.322"
    Rectangle (33,327 180x38), "SP_Lux: %.0f", text variable: P_Rum_4_322.fbLys.fbLightCtrl.fLuxZone1
    Button (45,96 150x30), "Top Button"
        tap P_Rum_4_322.bTopButtonZone1_Visu
    Button (45,136 150x30), "Bottom Button"
        tap P_Rum_4_322.bBottomButtonZone1_Visu
    Ellipse (46,187 22x23), colour toggle: P_Rum_4_322.fbLys.fbLightCtrl.bOnZone1
    Rectangle (78,187 122x22), "Lys Rum"
    Rectangle (46,252 71x22), "Dim Up", colour toggle: P_Rum_4_322.fbLys.fbLightCtrl.bDimUp
    Rectangle (127,252 71x22), "Dim Dwn", colour toggle: P_Rum_4_322.fbLys.fbLightCtrl.bDimDwn
    Ellipse (45,219 22x23), colour toggle: P_Rum_4_322.fbLys.fbLightCtrl.bAutoZone1
    Rectangle (78,219 122x22), "Lys Auto"
    Ellipse (45,54 22x23), colour toggle: P_Rum_4_322.fbLys.fbLightCtrl.bPIR
    Rectangle (77,54 122x22), "PIR status"
END_VISUALIZATION

// ---- POUs/Alle_Rum/Rum_Med_DALI_Pir/Rum_4_324/Visualization_4_324.TcVIS
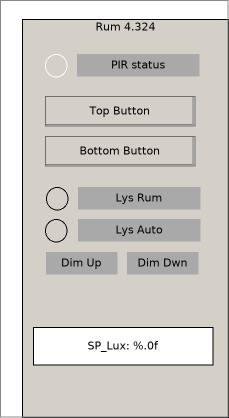
VISUALIZATION Visualization_4_324  // 229x418
    RoundedRectangle (22,19 207x399), "Rum 4.324"
    Rectangle (33,327 180x38), "SP_Lux: %.0f", text variable: P_Rum_4_324.fbLys.fbLightCtrl.fLuxZone1
    Button (45,96 150x30), "Top Button"
        tap P_Rum_4_324.bTopButtonZone1_Visu
    Button (45,136 150x30), "Bottom Button"
        tap P_Rum_4_324.bBottomButtonZone1_Visu
    Ellipse (46,187 22x23), colour toggle: P_Rum_4_324.fbLys.fbLightCtrl.bOnZone1
    Rectangle (78,187 122x22), "Lys Rum"
    Rectangle (46,252 71x22), "Dim Up", colour toggle: P_Rum_4_324.fbLys.fbLightCtrl.bDimUp
    Rectangle (127,252 71x22), "Dim Dwn", colour toggle: P_Rum_4_324.fbLys.fbLightCtrl.bDimDwn
    Ellipse (45,219 22x23), colour toggle: P_Rum_4_324.fbLys.fbLightCtrl.bAutoZone1
    Rectangle (78,219 122x22), "Lys Auto"
    Ellipse (45,54 22x23), colour toggle: P_Rum_4_324.fbLys.fbLightCtrl.bPIR
    Rectangle (77,54 122x22), "PIR status"
END_VISUALIZATION

// ---- POUs/Alle_Rum/Rum_Med_DALI_Pir/Rum_5_345/Visualization_5_345.TcVIS
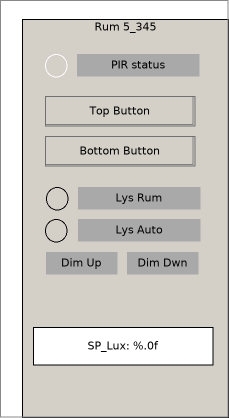
VISUALIZATION Visualization_5_345  // 229x418
    RoundedRectangle (22,19 207x399), "Rum 5_345"
    Rectangle (33,327 180x38), "SP_Lux: %.0f", text variable: P_Rum_5_345.fbLys.fbLightCtrl.fLuxZone1
    Button (45,96 150x30), "Top Button"
        tap P_Rum_5_345.bTopButtonZone1_Visu
    Button (45,136 150x30), "Bottom Button"
        tap P_Rum_5_345.bBottomButtonZone1_Visu
    Ellipse (46,187 22x23), colour toggle: P_Rum_5_345.fbLys.fbLightCtrl.bOnZone1
    Rectangle (78,187 122x22), "Lys Rum"
    Rectangle (46,252 71x22), "Dim Up", colour toggle: P_Rum_5_345.fbLys.fbLightCtrl.bDimUp
    Rectangle (127,252 71x22), "Dim Dwn", colour toggle: P_Rum_5_345.fbLys.fbLightCtrl.bDimDwn
    Ellipse (45,219 22x23), colour toggle: P_Rum_5_345.fbLys.fbLightCtrl.bAutoZone1
    Rectangle (78,219 122x22), "Lys Auto"
    Ellipse (45,54 22x23), colour toggle: P_Rum_5_345.fbLys.fbLightCtrl.bPIR
    Rectangle (77,54 122x22), "PIR status"
END_VISUALIZATION

// ---- POUs/Alle_Rum/Rum_Med_DALI_Pir/Rum_5_354/Visualization_5_354.TcVIS
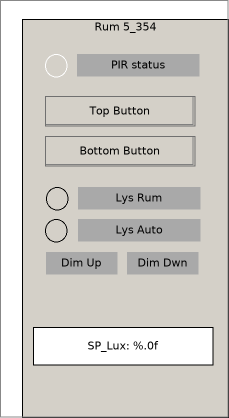
VISUALIZATION Visualization_5_354  // 229x418
    RoundedRectangle (22,19 207x399), "Rum 5_354"
    Rectangle (33,327 180x38), "SP_Lux: %.0f", text variable: P_Rum_4_324.fbLys.fbLightCtrl.fLuxZone1
    Button (45,96 150x30), "Top Button"
        tap P_Rum_5_354.bTopButtonZone1_Visu
    Button (45,136 150x30), "Bottom Button"
        tap P_Rum_5_354.bBottomButtonZone1_Visu
    Ellipse (46,187 22x23), colour toggle: P_Rum_5_354.fbLys.fbLightCtrl.bOnZone1
    Rectangle (78,187 122x22), "Lys Rum"
    Rectangle (46,252 71x22), "Dim Up", colour toggle: P_Rum_5_354.fbLys.fbLightCtrl.bDimUp
    Rectangle (127,252 71x22), "Dim Dwn", colour toggle: P_Rum_5_354.fbLys.fbLightCtrl.bDimDwn
    Ellipse (45,219 22x23), colour toggle: P_Rum_5_354.fbLys.fbLightCtrl.bAutoZone1
    Rectangle (78,219 122x22), "Lys Auto"
    Ellipse (45,54 22x23), colour toggle: P_Rum_5_354.fbLys.fbLightCtrl.bPIR
    Rectangle (77,54 122x22), "PIR status"
END_VISUALIZATION

// ---- POUs/Alle_Rum/Rum_Med_DALI_Pir/Rum_5_355A/Visualization_5_354_1.TcVIS
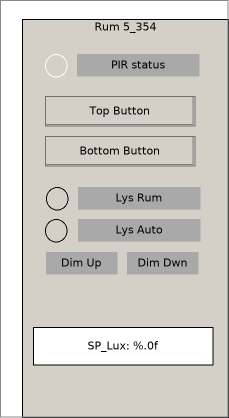
VISUALIZATION Visualization_5_354_1  // 229x418
    RoundedRectangle (22,19 207x399), "Rum 5_354"
    Rectangle (33,327 180x38), "SP_Lux: %.0f", text variable: P_Rum_4_324.fbLys.fbLightCtrl.fLuxZone1
    Button (45,96 150x30), "Top Button"
        tap P_Rum_5_354.bTopButtonZone1_Visu
    Button (45,136 150x30), "Bottom Button"
        tap P_Rum_5_354.bBottomButtonZone1_Visu
    Ellipse (46,187 22x23), colour toggle: P_Rum_5_354.fbLys.fbLightCtrl.bOnZone1
    Rectangle (78,187 122x22), "Lys Rum"
    Rectangle (46,252 71x22), "Dim Up", colour toggle: P_Rum_5_354.fbLys.fbLightCtrl.bDimUp
    Rectangle (127,252 71x22), "Dim Dwn", colour toggle: P_Rum_5_354.fbLys.fbLightCtrl.bDimDwn
    Ellipse (45,219 22x23), colour toggle: P_Rum_5_354.fbLys.fbLightCtrl.bAutoZone1
    Rectangle (78,219 122x22), "Lys Auto"
    Ellipse (45,54 22x23), colour toggle: P_Rum_5_354.fbLys.fbLightCtrl.bPIR
    Rectangle (77,54 122x22), "PIR status"
END_VISUALIZATION

// ---- POUs/DALI/DALI_Setup/VISUs/TextLists/EventPriority.TcTLO
TEXTLIST EventPriority
  2 = 'MiddleHigh'
  3 = 'Middle'
  4 = 'MiddleLow'
  5 = 'Low'
  255 = 'Unknown'
   = ''
END_TEXTLIST

// ---- POUs/DALI/DALI_Setup/VISUs/TextLists/ExtendedFadeTime.TcTLO
TEXTLIST ExtendedFadeTime
  0 = 'No Fade'
  1 = '1 * 100 ms = 100 ms'
  2 = '2 * 100 ms = 200 ms'
  3 = '3 * 100 ms = 300 ms'
  4 = '4 * 100 ms = 400 ms'
  5 = '5 * 100 ms = 500 ms'
  6 = '6 * 100 ms = 600 ms'
  7 = '7 * 100 ms = 700 ms'
  8 = '8 * 100 ms = 800 ms'
  9 = '9 * 100 ms = 900 ms'
  10 = '10 * 100 ms = 1000 ms'
  11 = '11 * 100 ms = 1100 ms'
  12 = '12 * 100 ms = 1200 ms'
  13 = '13 * 100 ms = 1300 ms'
  14 = '14 * 100 ms = 1400 ms'
  15 = '15 * 100 ms = 1500 ms'
  16 = '16 * 100 ms = 1600 ms'
  17 = '1 * 1 s = 1 s'
  18 = '2 * 1 s = 2 s'
  19 = '3 * 1 s = 3 s'
  20 = '4 * 1 s = 4 s'
  21 = '5 * 1 s = 5 s'
  22 = '6 * 1 s = 6 s'
  23 = '7 * 1 s = 7 s'
  24 = '8 * 1 s = 8 s'
  25 = '9 * 1 s = 9 s'
  26 = '10 * 1 s = 10 s'
  27 = '11 * 1 s = 11 s'
  28 = '12 * 1 s = 12 s'
  29 = '13 * 1 s = 13 s'
  30 = '14 * 1 s = 14 s'
  31 = '15 * 1 s = 15 s'
  32 = '16 * 1 s = 16 s'
  33 = '1 * 10 s = 10 s'
  34 = '2 * 10 s = 20 s'
  35 = '3 * 10 s = 30 s'
  36 = '4 * 10 s = 40 s'
  37 = '5 * 10 s = 50 s'
  38 = '6 * 10 s = 60 s'
  39 = '7 * 10 s = 70 s'
  40 = '8 * 10 s = 80 s'
  41 = '9 * 10 s = 90 s'
  42 = '10 * 10 s = 100 s'
  43 = '11 * 10 s = 110 s'
  44 = '12 * 10 s = 120 s'
  45 = '13 * 10 s = 130 s'
  46 = '14 * 10 s = 140 s'
  47 = '15 * 10 s = 150 s'
  48 = '16 * 10 s = 160 s'
  49 = '1 * 1 min = 1 min'
  50 = '2 * 1 min = 2 min'
  51 = '3 * 1 min = 3 min'
  52 = '4 * 1 min = 4 min'
  53 = '5 * 1 min = 5 min'
  54 = '6 * 1 min = 6 min'
  55 = '7 * 1 min = 7 min'
  56 = '8 * 1 min = 8 min'
  57 = '9 * 1 min = 9 min'
  58 = '10 * 1 min = 10 min'
  59 = '11 * 1 min = 11 min'
  60 = '12 * 1 min = 12 min'
  61 = '13 * 1 min = 13 min'
  62 = '14 * 1 min = 14 min'
  63 = '15 * 1 min = 15 min'
  64 = '16 * 1 min = 16 min'
  255 = 'Unknown'
   = ''
END_TEXTLIST

// ---- POUs/DALI/DALI_Setup/VISUs/TextLists/FadeRate.TcTLO
TEXTLIST FadeRate
  0 = 'Unknown'
  1 = '358 steps/s'
  2 = '253 steps/s'
  3 = '179 steps/s'
  4 = '127 steps/s'
  5 = '89,4 steps/s'
  6 = '63,3 steps/s'
  7 = '44,7 steps/s'
  8 = '31,6 steps/s'
  9 = '22,4 steps/s'
  10 = '15,8 steps/s'
  11 = '11,2 steps/s'
  12 = '7,9 steps/s'
  13 = '5,6 steps/s'
  14 = '4,0 steps/s'
  15 = '2,8 steps/s'
  255 = 'Unknown'
   = ''
END_TEXTLIST

// ---- POUs/DALI/DALI_Setup/VISUs/TextLists/FastFadeTime.TcTLO
TEXTLIST FastFadeTime
  0 = 'Disabled'
  4 = 'T100ms'
  8 = 'T200ms'
  12 = 'T300ms'
  16 = 'T400ms'
  20 = 'T500ms'
  24 = 'T600ms'
  27 = 'T700ms'
  255 = 'Unknown'
   = ''
END_TEXTLIST

// ---- POUs/DALI/DALI_Setup/VISUs/TextLists/TextList_Dialogs.TcTLO
TEXTLIST TextList_Dialogs
  0 = 'Select the function'
  1 = 'Control Gears - Commands'
  2 = 'Control Gears - Addressing'
  3 = 'Control Gears - Parameters'
  4 = 'Control Gears - Groups'
  5 = 'Control Gears - Scenes'
  6 = 'Control Gears - Memory Pages'
  7 = 'Control Gears - Set Fading'
  8 = 'Control Gears - Device Type 1 (Emergency lighting)'
  9 = 'Control Gears - Device Type 4 (Incandescent lamp)'
  10 = 'Control Gears - Device Type 6 (LED)'
  11 = 'Control Gears - Device Type 7 (Switching)'
  12 = 'Control Devices - Addressing'
  13 = 'Control Devices - Parameters'
  15 = 'Control Devices - Device Type 1 (Push button)'
  16 = 'Control Devices - Device Type 2 (Absolute input)'
  17 = 'Control Devices - Device Type 3 (Occupancy sensor)'
  18 = 'Control Devices - Device Type 4 (Light sensor)'
  19 = 'Control Devices - Device Type 0 (Generic instance)'
  20 = 'Control Devices - Memory Pages'
  14 = 'Control Devices - Identify'
   = ''
END_TEXTLIST

// ---- POUs/DALI/DALI_Setup/VISUs/Visu_DALICommissioning/Visu_Part102Commands.TcVIS
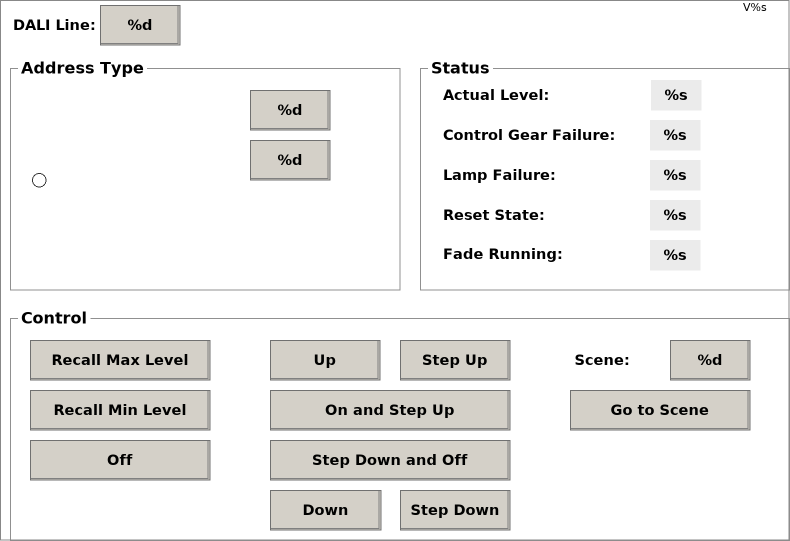
VISUALIZATION Visu_Part102Commands  // 790x541
    GroupBox (10,310 780x231), "Control"
        Button (20,130 180x40), "Off"
            OnMouseClick: execute { DALI_Commissioning.fbPart102Commands.bOff := TRUE; }
        Button (20,80 180x40), "Recall Min Level"
            OnMouseClick: execute { DALI_Commissioning.fbPart102Commands.bRecallMinLevel := TRUE; }
        Button (20,30 180x40), "Recall Max Level"
            OnMouseClick: execute { DALI_Commissioning.fbPart102Commands.bRecallMaxLevel := TRUE; }
        Button (260,180 111x40), "Down"
            OnMouseClick: execute { DALI_Commissioning.fbPart102Commands.bDown := TRUE; }
        Button (390,180 110x40), "Step Down"
            OnMouseClick: execute { DALI_Commissioning.fbPart102Commands.bStepDown := TRUE; }
        Button (260,130 240x40), "Step Down and Off"
            OnMouseClick: execute { DALI_Commissioning.fbPart102Commands.bStepDownAndOff := TRUE; }
        Button (660,30 80x40), "%d", text variable: DALI_Commissioning.fbPart102Commands.nScene
            OnMouseClick: write the text variable via Default, min 0, max 15, title "Insert scene number"
        Textfield (550,35 85x30), "Scene:"
        Button (560,80 180x40), "Go to Scene"
            OnMouseClick: execute { DALI_Commissioning.fbPart102Commands.bGotoScene := TRUE; }
        Button (260,80 240x40), "On and Step Up"
            OnMouseClick: execute { DALI_Commissioning.fbPart102Commands.bOnAndStepUp := TRUE; }
        Button (260,30 110x40), "Up"
            OnMouseClick: execute { DALI_Commissioning.fbPart102Commands.bUp := TRUE; }
        Button (390,30 110x40), "Step Up"
            OnMouseClick: execute { DALI_Commissioning.fbPart102Commands.bStepUp := TRUE; }
    GroupBox (420,60 370x230), "Status"
        Textfield (20,20 200x30), "Actual Level:"
        Textfield (20,60 200x30), "Control Gear Failure:"
        Textfield (231,20 50x30), "%s", text variable: DALI_Commissioning.fbPart102Commands.sActualLevel
        Textfield (230,60 50x30), "%s", text variable: DALI_Commissioning.fbPart102Commands.sControlGearFailure
        Textfield (20,100 200x30), "Lamp Failure:"
        Textfield (230,100 50x30), "%s", text variable: DALI_Commissioning.fbPart102Commands.sLampFailure
        Textfield (20,140 200x30), "Reset State:"
        Textfield (230,140 50x30), "%s", text variable: DALI_Commissioning.fbPart102Commands.sResetState
        Textfield (20,180 200x28), "Fade Running:"
        Textfield (230,180 50x30), "%s", text variable: DALI_Commissioning.fbPart102Commands.sFadeRunning
    GroupBox (10,60 390x230), "Address Type"
        Button (240,30 80x40), "%d", text variable: DALI_Commissioning.fbPart102Commands.nShortAddress
            OnMouseClick: write the text variable via Default, min 0, max 63, title "Insert Short Address"
            OnMouseClick: execute {  }
        RadioButton (20,20 190x200), variable: DALI_Commissioning.fbPart102Commands.eAddressType
            Areas[0]: Text=Short Address
            Areas[1]: Text=Group Address
            Areas[2]: Text=Broadcast
            Areas[3]: Text=Unaddressed
        Button (240,80 80x40), "%d", text variable: DALI_Commissioning.fbPart102Commands.nGroupAddress
            OnMouseClick: write the text variable via Default, min 0, max 15, title "Insert Group Address"
    Rectangle (720,0 70x15), "V%s", text variable: stLibVersion_Tc3_DALI_PLC_Commissioning_Tool.sVersion
    Group (10,5 170x40)
        Textfield (0,0 110x40), "DALI Line:"
        Button (90,0 80x40), "%d", text variable: GVL_Internal.nDALILine
            OnMouseClick: write the text variable via Default, min 1, max 10, title "Choose line"
END_VISUALIZATION

// ---- POUs/DALI/DALI_Setup/VISUs/Visu_DALICommissioning/Visu_Part103MemoryBank.TcVIS
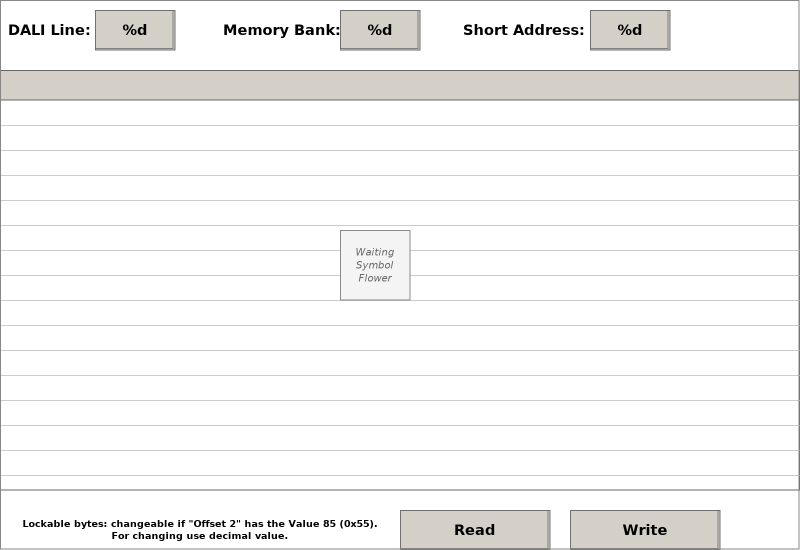
VISUALIZATION Visu_Part103MemoryBank  // 800x550
    Table (0,70 800x420), data array: DALI_Commissioning.fbPart103MemoryPages.aMemoryBank
        p3854506369: DALI_Commissioning.fbPart103MemoryPages.aMemoryBank[INDEX].sOffset
        p1892666644: DALI_Commissioning.fbPart103MemoryPages.aMemoryBank[INDEX].sName
        p338671338: DALI_Commissioning.fbPart103MemoryPages.aMemoryBank[INDEX].nValueDec
        p2170511999: DALI_Commissioning.fbPart103MemoryPages.aMemoryBank[INDEX].nValueHex
        p1755163831: Value Dec
        p4092479075: Value Hex
        p1137915858: DALI_Commissioning.fbPart103MemoryPages.nOffset
        Columns.Column.[0].Template: DALI_Commissioning.fbPart103MemoryPages.aNoValue[INDEX]
        Columns.Column.[1].Template: DALI_Commissioning.fbPart103MemoryPages.aNoValue[INDEX]
        Columns.Column.[2].Template: DALI_Commissioning.fbPart103MemoryPages.aNoValue[INDEX]; DALI_Commissioning.fbPart103MemoryPages.nMemoryBank=0; OnMouseClick: write the text variable via Default, min 0, max 255, title "Lockable variable decimal"
        Columns.Column.[3].Template: DALI_Commissioning.fbPart103MemoryPages.aNoValue[INDEX]; OnMouseClick: write the text variable via Default, title "Lockable variable hexadecimal"
    Button (400,510 150x40), "Read"
        OnMouseClick: execute { DALI_Commissioning.fbPart103MemoryPages.bRead := TRUE; }
    Button (570,510 150x40), "Write"
        OnMouseClick: execute { DALI_Commissioning.fbPart103MemoryPages.bWrite := TRUE; }
    Textfield (15,510 370x40), "Lockable bytes: changeable if "Offset 2" has the Value 85 (0x55). For changing use decimal value."
    WaitingSymbolFlower (340,230 70x70), invisible if: DALI_Commissioning.fbPart103MemoryPages.bHideWaitSymbol
    Textfield (460,10 130x40), "Short Address:"
    Button (590,10 80x40), "%d", text variable: DALI_Commissioning.fbPart103MemoryPages.nAddress
        OnMouseClick: write the text variable via Default, min 0, max 63, title "Insert Short Address"
    Group (220,10 200x40)
        Textfield (0,0 150x40), "Memory Bank:"
        Button (120,0 80x40), "%d", text variable: DALI_Commissioning.fbPart103MemoryPages.nMemoryBank
            OnMouseClick: write the text variable via Default, min 0, max 255, title "Insert Memory Bank"
    Group (5,10 170x40)
        Textfield (0,0 110x40), "DALI Line:"
        Button (90,0 80x40), "%d", text variable: GVL_Internal.nDALILine
            OnMouseClick: write the text variable via Default, min 1, max 10, title "Choose line"
END_VISUALIZATION

// ---- POUs/DALI/DALI_Setup/VISUs/Visu_DALICommissioning/Visu_Part103Parameters.TcVIS
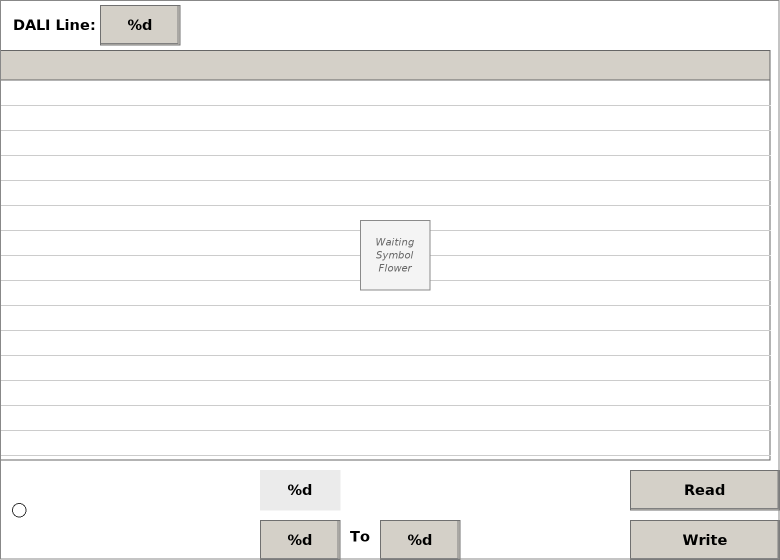
VISUALIZATION Visu_Part103Parameters  // 780x560
    Table (0,50 770x410), data array: DALI_Commissioning.fbPart103Parameters.aParameters
        p1137915858: DALI_Commissioning.fbPart103Parameters.nSelectedAddress
        p3854506369: DALI_Commissioning.fbPart103Parameters.aParameters[INDEX].nOperatingMode
        p1892666644: DALI_Commissioning.fbPart103Parameters.aParameters[INDEX].sInstanceType0
        p338671338: DALI_Commissioning.fbPart103Parameters.aParameters[INDEX].sInstanceType1
        p2170511999: DALI_Commissioning.fbPart103Parameters.aParameters[INDEX].sInstanceType2
        p3723444502: DALI_Commissioning.fbPart103Parameters.aParameters[INDEX].sInstanceType3
        p1218418051: DALI_Commissioning.fbPart103Parameters.aParameters[INDEX].sInstanceType4
        p511219082: IT0 (Generic Input)
        p1755163831: IT1 (PushButton)
        p4092479075: IT2 (Absolute Input)
        p2237128397: IT3 (Occupancy)
        p505689113: IT4 (Light Sensor)
        Columns.Column.[0].Template: OnMouseClick: write the text variable via Default, min 0, max 255, title "Insert Operating Mode 0, 128-255"
    RadioButton (10,460 230x100), variable: DALI_Commissioning.fbPart103Parameters.nAddressRange
        Areas[0]: Text=Single Short Address
        Areas[1]: Text=Short Address Range
    Textfield (260,470 80x40), "%d", text variable: DALI_Commissioning.fbPart103Parameters.nSelectedAddress
    Button (260,520 80x40), "%d", text variable: DALI_Commissioning.fbPart103Parameters.nStartAddress
        OnMouseClick: write the text variable via Default, min 0, max 63, title "Insert Short Address"
    Button (380,520 80x40), "%d", text variable: DALI_Commissioning.fbPart103Parameters.nEndAddress
        OnMouseClick: write the text variable via Default, min 0, max 63, title "Insert Short Address"
    Button (630,470 150x40), "Read"
        OnMouseClick: execute { DALI_Commissioning.fbPart103Parameters.bRead := true; }
    Button (630,520 150x40), "Write"
        OnMouseClick: execute { DALI_Commissioning.fbPart103Parameters.bWrite := true; }
    Textfield (335,521 50x31), "To"
    WaitingSymbolFlower (360,220 70x70), invisible if: DALI_Commissioning.fbPart103Parameters.bHideWaitSymbol
    Group (10,5 170x40)
        Textfield (0,0 110x40), "DALI Line:"
        Button (90,0 80x40), "%d", text variable: GVL_Internal.nDALILine
            OnMouseClick: write the text variable via Default, min 1, max 10, title "Choose line"
END_VISUALIZATION

// ---- POUs/DALI/DALI_Setup/VISUs/Visu_DALICommissioning/Visu_Part202.TcVIS
